   1:  PR[91,1] = PR[90,1] + -40.639;
   1:  PR[91,2] = PR[90,2] + 3.831;
   1:L PR[91] R[100]mm/sec CNT100;
   1:  PR[91,1] = PR[90,1] + -40.703;
   1:  PR[91,2] = PR[90,2] + 3.535;
   1:L PR[91] R[100]mm/sec CNT100;
   1:  PR[91,1] = PR[90,1] + -40.740;
   1:  PR[91,2] = PR[90,2] + 3.017;
   1:L PR[91] R[100]mm/sec CNT100;
   1:  PR[91,1] = PR[90,1] + -41.147;
   1:  PR[91,2] = PR[90,2] + -0.477;
   1:L PR[91] R[100]mm/sec CNT100;
   1:  PR[91,1] = PR[90,1] + -41.119;
   1:  PR[91,2] = PR[90,2] + -0.869;
   1:L PR[91] R[100]mm/sec CNT100;
   1:  PR[91,1] = PR[90,1] + -40.715;
   1:  PR[91,2] = PR[90,2] + -4.331;
   1:L PR[91] R[100]mm/sec CNT100;
   1:  PR[91,1] = PR[90,1] + -40.638;
   1:  PR[91,2] = PR[90,2] + -4.679;
   1:L PR[91] R[100]mm/sec CNT100;
   1:  PR[91,1] = PR[90,1] + -39.266;
   1:  PR[91,2] = PR[90,2] + -8.416;
   1:L PR[91] R[100]mm/sec CNT100;
   1:  PR[91,1] = PR[90,1] + -39.110;
   1:  PR[91,2] = PR[90,2] + -8.700;
   1:L PR[91] R[100]mm/sec CNT100;
   1:  PR[91,1] = PR[90,1] + -37.111;
   1:  PR[91,2] = PR[90,2] + -11.734;
   1:L PR[91] R[100]mm/sec CNT100;
   1:  PR[91,1] = PR[90,1] + -36.935;
   1:  PR[91,2] = PR[90,2] + -11.967;
   1:L PR[91] R[100]mm/sec CNT100;
   1:  PR[91,1] = PR[90,1] + -36.697;
   1:  PR[91,2] = PR[90,2] + -12.203;
   1:L PR[91] R[100]mm/sec CNT100;
   1:  PR[91,1] = PR[90,1] + -33.985;
   1:  PR[91,2] = PR[90,2] + -14.753;
   1:L PR[91] R[100]mm/sec CNT100;
   1:  PR[91,1] = PR[90,1] + -33.873;
   1:  PR[91,2] = PR[90,2] + -14.836;
   1:L PR[91] R[100]mm/sec CNT100;
   1:  PR[91,1] = PR[90,1] + -33.596;
   1:  PR[91,2] = PR[90,2] + -14.985;
   1:L PR[91] R[100]mm/sec CNT100;
   1:  PR[91,1] = PR[90,1] + -30.271;
   1:  PR[91,2] = PR[90,2] + -16.901;
   1:L PR[91] R[100]mm/sec CNT100;
   1:  PR[91,1] = PR[90,1] + -30.216;
   1:  PR[91,2] = PR[90,2] + -16.922;
   1:L PR[91] R[100]mm/sec CNT100;
   1:  PR[91,1] = PR[90,1] + -26.322;
   1:  PR[91,2] = PR[90,2] + -18.082;
   1:L PR[91] R[100]mm/sec CNT100;
   1:  PR[91,1] = PR[90,1] + -22.141;
   1:  PR[91,2] = PR[90,2] + -18.325;
   1:L PR[91] R[100]mm/sec CNT100;
   1:  PR[91,1] = PR[90,1] + -17.967;
   1:  PR[91,2] = PR[90,2] + -17.608;
   1:L PR[91] R[100]mm/sec CNT100;
   1:  PR[91,1] = PR[90,1] + -14.146;
   1:  PR[91,2] = PR[90,2] + -15.991;
   1:L PR[91] R[100]mm/sec CNT100;
   1:  PR[91,1] = PR[90,1] + -13.906;
   1:  PR[91,2] = PR[90,2] + -15.838;
   1:L PR[91] R[100]mm/sec CNT100;
   1:  PR[91,1] = PR[90,1] + -10.813;
   1:  PR[91,2] = PR[90,2] + -13.575;
   1:L PR[91] R[100]mm/sec CNT100;
   1:  PR[91,1] = PR[90,1] + -10.403;
   1:  PR[91,2] = PR[90,2] + -13.158;
   1:L PR[91] R[100]mm/sec CNT100;
   1:  PR[91,1] = PR[90,1] + -8.128;
   1:  PR[91,2] = PR[90,2] + -10.487;
   1:L PR[91] R[100]mm/sec CNT100;
   1:  PR[91,1] = PR[90,1] + -7.743;
   1:  PR[91,2] = PR[90,2] + -9.851;
   1:L PR[91] R[100]mm/sec CNT100;
   1:  PR[91,1] = PR[90,1] + -9.545;
   1:  PR[91,2] = PR[90,2] + -9.686;
   1:L PR[91] R[100]mm/sec CNT100;
   1:  PR[91,1] = PR[90,1] + -5.350;
   1:  PR[91,2] = PR[90,2] + -5.740;
   1:L PR[91] R[100]mm/sec CNT100;
   1:  PR[91,1] = PR[90,1] + -5.315;
   1:  PR[91,2] = PR[90,2] + -5.719;
   1:L PR[91] R[100]mm/sec CNT100;
   1:  PR[91,1] = PR[90,1] + -4.925;
   1:  PR[91,2] = PR[90,2] + -5.085;
   1:L PR[91] R[100]mm/sec CNT100;
   1:  PR[91,1] = PR[90,1] + -2.728;
   1:  PR[91,2] = PR[90,2] + -4.248;
   1:L PR[91] R[100]mm/sec CNT100;
   1:  PR[91,1] = PR[90,1] + 2.325;
   1:L PR[91] R[100]mm/sec CNT100;
   1:  PR[91,1] = PR[90,1] + 3.225;
   1:  PR[91,2] = PR[90,2] + -4.625;
   1:L PR[91] R[100]mm/sec CNT100;
   1:  PR[91,1] = PR[90,1] + 4.250;
   1:  PR[91,2] = PR[90,2] + -5.004;
   1:L PR[91] R[100]mm/sec CNT100;
   1:  PR[91,1] = PR[90,1] + 4.835;
   1:  PR[91,2] = PR[90,2] + -5.693;
   1:L PR[91] R[100]mm/sec CNT100;
   1:  PR[91,1] = PR[90,1] + 4.918;
   1:  PR[91,2] = PR[90,2] + -5.761;
   1:L PR[91] R[100]mm/sec CNT100;
   1:  PR[91,1] = PR[90,1] + 5.507;
   1:  PR[91,2] = PR[90,2] + -6.410;
   1:L PR[91] R[100]mm/sec CNT100;
   1:  PR[91,1] = PR[90,1] + 7.186;
   1:  PR[91,2] = PR[90,2] + -9.719;
   1:L PR[91] R[100]mm/sec CNT100;
   1:  PR[91,1] = PR[90,1] + 7.651;
   1:  PR[91,2] = PR[90,2] + -10.488;
   1:L PR[91] R[100]mm/sec CNT100;
   1:  PR[91,1] = PR[90,1] + 9.927;
   1:  PR[91,2] = PR[90,2] + -13.160;
   1:L PR[91] R[100]mm/sec CNT100;
   1:  PR[91,1] = PR[90,1] + 10.337;
   1:  PR[91,2] = PR[90,2] + -13.578;
   1:L PR[91] R[100]mm/sec CNT100;
   1:  PR[91,1] = PR[90,1] + 13.428;
   1:  PR[91,2] = PR[90,2] + -15.840;
   1:L PR[91] R[100]mm/sec CNT100;
   1:  PR[91,1] = PR[90,1] + 13.668;
   1:  PR[91,2] = PR[90,2] + -15.992;
   1:L PR[91] R[100]mm/sec CNT100;
   1:  PR[91,1] = PR[90,1] + 17.491;
   1:  PR[91,2] = PR[90,2] + -17.609;
   1:L PR[91] R[100]mm/sec CNT100;
   1:  PR[91,1] = PR[90,1] + 21.626;
   1:  PR[91,2] = PR[90,2] + -18.322;
   1:L PR[91] R[100]mm/sec CNT100;
   1:  PR[91,1] = PR[90,1] + 25.845;
   1:  PR[91,2] = PR[90,2] + -18.081;
   1:L PR[91] R[100]mm/sec CNT100;
   1:  PR[91,1] = PR[90,1] + 29.738;
   1:  PR[91,2] = PR[90,2] + -16.921;
   1:L PR[91] R[100]mm/sec CNT100;
   1:  PR[91,1] = PR[90,1] + 29.796;
   1:  PR[91,2] = PR[90,2] + -16.899;
   1:L PR[91] R[100]mm/sec CNT100;
   1:  PR[91,1] = PR[90,1] + 33.369;
   1:  PR[91,2] = PR[90,2] + -14.854;
   1:L PR[91] R[100]mm/sec CNT100;
   1:  PR[91,1] = PR[90,1] + 33.480;
   1:  PR[91,2] = PR[90,2] + -14.772;
   1:L PR[91] R[100]mm/sec CNT100;
   1:  PR[91,1] = PR[90,1] + 33.701;
   1:  PR[91,2] = PR[90,2] + -14.553;
   1:L PR[91] R[100]mm/sec CNT100;
   1:  PR[91,1] = PR[90,1] + 36.475;
   1:  PR[91,2] = PR[90,2] + -11.941;
   1:L PR[91] R[100]mm/sec CNT100;
   1:  PR[91,1] = PR[90,1] + 36.631;
   1:  PR[91,2] = PR[90,2] + -11.732;
   1:L PR[91] R[100]mm/sec CNT100;
   1:  PR[91,1] = PR[90,1] + 38.630;
   1:  PR[91,2] = PR[90,2] + -8.699;
   1:L PR[91] R[100]mm/sec CNT100;
   1:  PR[91,1] = PR[90,1] + 38.791;
   1:  PR[91,2] = PR[90,2] + -8.407;
   1:L PR[91] R[100]mm/sec CNT100;
   1:  PR[91,1] = PR[90,1] + 38.939;
   1:  PR[91,2] = PR[90,2] + -8.013;
   1:L PR[91] R[100]mm/sec CNT100;
   1:  PR[91,1] = PR[90,1] + 40.159;
   1:  PR[91,2] = PR[90,2] + -4.682;
   1:L PR[91] R[100]mm/sec CNT100;
   1:  PR[91,1] = PR[90,1] + 40.223;
   1:  PR[91,2] = PR[90,2] + -4.386;
   1:L PR[91] R[100]mm/sec CNT100;
   1:  PR[91,1] = PR[90,1] + 40.261;
   1:  PR[91,2] = PR[90,2] + -3.867;
   1:L PR[91] R[100]mm/sec CNT100;
   1:  PR[91,1] = PR[90,1] + 40.667;
   1:  PR[91,2] = PR[90,2] + -0.370;
   1:L PR[91] R[100]mm/sec CNT100;
   1:  PR[91,1] = PR[90,1] + 40.639;
   1:  PR[91,2] = PR[90,2] + 0.022;
   1:L PR[91] R[100]mm/sec CNT100;
   1:  PR[91,1] = PR[90,1] + 40.235;
   1:  PR[91,2] = PR[90,2] + 3.486;
   1:L PR[91] R[100]mm/sec CNT100;
   1:  PR[91,1] = PR[90,1] + 40.159;
   1:  PR[91,2] = PR[90,2] + 3.833;
   1:L PR[91] R[100]mm/sec CNT100;
   1:  PR[91,1] = PR[90,1] + 38.787;
   1:  PR[91,2] = PR[90,2] + 7.567;
   1:L PR[91] R[100]mm/sec CNT100;
   1:  PR[91,1] = PR[90,1] + 38.631;
   1:  PR[91,2] = PR[90,2] + 7.852;
   1:L PR[91] R[100]mm/sec CNT100;
   1:  PR[91,1] = PR[90,1] + 36.632;
   1:  PR[91,2] = PR[90,2] + 10.885;
   1:L PR[91] R[100]mm/sec CNT100;
   1:  PR[91,1] = PR[90,1] + 36.456;
   1:  PR[91,2] = PR[90,2] + 11.118;
   1:L PR[91] R[100]mm/sec CNT100;
   1:  PR[91,1] = PR[90,1] + 36.218;
   1:  PR[91,2] = PR[90,2] + 11.354;
   1:L PR[91] R[100]mm/sec CNT100;
   1:  PR[91,1] = PR[90,1] + 33.507;
   1:  PR[91,2] = PR[90,2] + 13.905;
   1:L PR[91] R[100]mm/sec CNT100;
   1:  PR[91,1] = PR[90,1] + 33.394;
   1:  PR[91,2] = PR[90,2] + 13.989;
   1:L PR[91] R[100]mm/sec CNT100;
   1:  PR[91,1] = PR[90,1] + 33.118;
   1:  PR[91,2] = PR[90,2] + 14.138;
   1:L PR[91] R[100]mm/sec CNT100;
   1:  PR[91,1] = PR[90,1] + 29.794;
   1:  PR[91,2] = PR[90,2] + 16.053;
   1:L PR[91] R[100]mm/sec CNT100;
   1:  PR[91,1] = PR[90,1] + 29.738;
   1:  PR[91,2] = PR[90,2] + 16.073;
   1:L PR[91] R[100]mm/sec CNT100;
   1:  PR[91,1] = PR[90,1] + 25.840;
   1:  PR[91,2] = PR[90,2] + 17.235;
   1:L PR[91] R[100]mm/sec CNT100;
   1:  PR[91,1] = PR[90,1] + 21.627;
   1:  PR[91,2] = PR[90,2] + 17.475;
   1:L PR[91] R[100]mm/sec CNT100;
   1:  PR[91,1] = PR[90,1] + 17.492;
   1:  PR[91,2] = PR[90,2] + 16.762;
   1:L PR[91] R[100]mm/sec CNT100;
   1:  PR[91,1] = PR[90,1] + 13.669;
   1:  PR[91,2] = PR[90,2] + 15.146;
   1:L PR[91] R[100]mm/sec CNT100;
   1:  PR[91,1] = PR[90,1] + 13.430;
   1:  PR[91,2] = PR[90,2] + 14.993;
   1:L PR[91] R[100]mm/sec CNT100;
   1:  PR[91,1] = PR[90,1] + 10.338;
   1:  PR[91,2] = PR[90,2] + 12.732;
   1:L PR[91] R[100]mm/sec CNT100;
   1:  PR[91,1] = PR[90,1] + 9.927;
   1:  PR[91,2] = PR[90,2] + 12.314;
   1:L PR[91] R[100]mm/sec CNT100;
   1:  PR[91,1] = PR[90,1] + 7.650;
   1:  PR[91,2] = PR[90,2] + 9.639;
   1:L PR[91] R[100]mm/sec CNT100;
   1:  PR[91,1] = PR[90,1] + 7.199;
   1:  PR[91,2] = PR[90,2] + 8.897;
   1:L PR[91] R[100]mm/sec CNT100;
   1:  PR[91,1] = PR[90,1] + 5.521;
   1:  PR[91,2] = PR[90,2] + 5.588;
   1:L PR[91] R[100]mm/sec CNT100;
   1:  PR[91,1] = PR[90,1] + 4.973;
   1:  PR[91,2] = PR[90,2] + 4.956;
   1:L PR[91] R[100]mm/sec CNT100;
   1:  PR[91,1] = PR[90,1] + 4.835;
   1:  PR[91,2] = PR[90,2] + 4.871;
   1:L PR[91] R[100]mm/sec CNT100;
   1:  PR[91,1] = PR[90,1] + 4.448;
   1:  PR[91,2] = PR[90,2] + 4.242;
   1:L PR[91] R[100]mm/sec CNT100;
   1:  PR[91,1] = PR[90,1] + 2.263;
   1:  PR[91,2] = PR[90,2] + 3.401;
   1:L PR[91] R[100]mm/sec CNT100;
   1:  PR[91] = PR[90];
   1:  PR[91,1] = PR[90,1] + -2.779;
   1:  PR[91,2] = PR[90,2] + 3.945;
   1:  PR[91,3] = PR[90,3] + 11.895;
   1:L PR[91] R[100]mm/sec CNT100;
   1:  PR[91,1] = PR[90,1] + -4.758;
   1:  PR[91,2] = PR[90,2] + 4.725;
   1:L PR[91] R[100]mm/sec CNT100;
   1:  PR[91,1] = PR[90,1] + -5.390;
   1:  PR[91,2] = PR[90,2] + 5.478;
   1:L PR[91] R[100]mm/sec CNT100;
   1:  PR[91,1] = PR[90,1] + -5.443;
   1:  PR[91,2] = PR[90,2] + 5.521;
   1:L PR[91] R[100]mm/sec CNT100;
   1:  PR[91,1] = PR[90,1] + -5.916;
   1:  PR[91,2] = PR[90,2] + 6.032;
   1:L PR[91] R[100]mm/sec CNT100;
   1:  PR[91,1] = PR[90,1] + -6.700;
   1:  PR[91,2] = PR[90,2] + 7.567;
   1:L PR[91] R[100]mm/sec CNT100;
   1:  PR[91,1] = PR[90,1] + -6.925;
   1:  PR[91,2] = PR[90,2] + 8.038;
   1:L PR[91] R[100]mm/sec CNT100;
   1:  PR[91,1] = PR[90,1] + -8.136;
   1:  PR[91,2] = PR[90,2] + 10.031;
   1:L PR[91] R[100]mm/sec CNT100;
   1:  PR[91,1] = PR[90,1] + -9.464;
   1:  PR[91,2] = PR[90,2] + 11.590;
   1:L PR[91] R[100]mm/sec CNT100;
   1:  PR[91,1] = PR[90,1] + -10.869;
   1:  PR[91,2] = PR[90,2] + 13.017;
   1:L PR[91] R[100]mm/sec CNT100;
   1:  PR[91,1] = PR[90,1] + -12.830;
   1:  PR[91,2] = PR[90,2] + 14.451;
   1:L PR[91] R[100]mm/sec CNT100;
   1:  PR[91,1] = PR[90,1] + -14.219;
   1:  PR[91,2] = PR[90,2] + 15.336;
   1:L PR[91] R[100]mm/sec CNT100;
   1:  PR[91,1] = PR[90,1] + -16.835;
   1:  PR[91,2] = PR[90,2] + 16.442;
   1:L PR[91] R[100]mm/sec CNT100;
   1:  PR[91,1] = PR[90,1] + -18.025;
   1:  PR[91,2] = PR[90,2] + 16.868;
   1:L PR[91] R[100]mm/sec CNT100;
   1:  PR[91,1] = PR[90,1] + -21.222;
   1:  PR[91,2] = PR[90,2] + 17.414;
   1:L PR[91] R[100]mm/sec CNT100;
   1:  PR[91,1] = PR[90,1] + -22.100;
   1:  PR[91,2] = PR[90,2] + 17.520;
   1:L PR[91] R[100]mm/sec CNT100;
   1:  PR[91,1] = PR[90,1] + -25.708;
   1:  PR[91,2] = PR[90,2] + 17.300;
   1:L PR[91] R[100]mm/sec CNT100;
   1:  PR[91,1] = PR[90,1] + -26.240;
   1:  PR[91,2] = PR[90,2] + 17.245;
   1:L PR[91] R[100]mm/sec CNT100;
   1:  PR[91,1] = PR[90,1] + -30.007;
   1:  PR[91,2] = PR[90,2] + 16.115;
   1:L PR[91] R[100]mm/sec CNT100;
   1:  PR[91,1] = PR[90,1] + -30.222;
   1:  PR[91,2] = PR[90,2] + 16.042;
   1:L PR[91] R[100]mm/sec CNT100;
   1:  PR[91,1] = PR[90,1] + -33.862;
   1:  PR[91,2] = PR[90,2] + 13.940;
   1:L PR[91] R[100]mm/sec CNT100;
   1:  PR[91,1] = PR[90,1] + -36.897;
   1:  PR[91,2] = PR[90,2] + 11.090;
   1:L PR[91] R[100]mm/sec CNT100;
   1:  PR[91,1] = PR[90,1] + -39.194;
   1:  PR[91,2] = PR[90,2] + 7.604;
   1:L PR[91] R[100]mm/sec CNT100;
   1:  PR[91,1] = PR[90,1] + -40.607;
   1:  PR[91,2] = PR[90,2] + 3.743;
   1:L PR[91] R[100]mm/sec CNT100;
   1:  PR[91,1] = PR[90,1] + -41.096;
   1:  PR[91,2] = PR[90,2] + -0.424;
   1:L PR[91] R[100]mm/sec CNT100;
   1:  PR[91,1] = PR[90,1] + -40.607;
   1:  PR[91,2] = PR[90,2] + -4.590;
   1:L PR[91] R[100]mm/sec CNT100;
   1:  PR[91,1] = PR[90,1] + -39.177;
   1:  PR[91,2] = PR[90,2] + -8.483;
   1:L PR[91] R[100]mm/sec CNT100;
   1:  PR[91,1] = PR[90,1] + -38.095;
   1:  PR[91,2] = PR[90,2] + -10.124;
   1:L PR[91] R[100]mm/sec CNT100;
   1:  PR[91,1] = PR[90,1] + -36.896;
   1:  PR[91,2] = PR[90,2] + -11.938;
   1:L PR[91] R[100]mm/sec CNT100;
   1:  PR[91,1] = PR[90,1] + -33.860;
   1:  PR[91,2] = PR[90,2] + -14.789;
   1:L PR[91] R[100]mm/sec CNT100;
   1:  PR[91,1] = PR[90,1] + -30.220;
   1:  PR[91,2] = PR[90,2] + -16.890;
   1:L PR[91] R[100]mm/sec CNT100;
   1:  PR[91,1] = PR[90,1] + -30.004;
   1:  PR[91,2] = PR[90,2] + -16.963;
   1:L PR[91] R[100]mm/sec CNT100;
   1:  PR[91,1] = PR[90,1] + -26.236;
   1:  PR[91,2] = PR[90,2] + -18.093;
   1:L PR[91] R[100]mm/sec CNT100;
   1:  PR[91,1] = PR[90,1] + -25.705;
   1:  PR[91,2] = PR[90,2] + -18.147;
   1:L PR[91] R[100]mm/sec CNT100;
   1:  PR[91,1] = PR[90,1] + -22.097;
   1:  PR[91,2] = PR[90,2] + -18.367;
   1:L PR[91] R[100]mm/sec CNT100;
   1:  PR[91,1] = PR[90,1] + -21.219;
   1:  PR[91,2] = PR[90,2] + -18.261;
   1:L PR[91] R[100]mm/sec CNT100;
   1:  PR[91,1] = PR[90,1] + -18.021;
   1:  PR[91,2] = PR[90,2] + -17.714;
   1:L PR[91] R[100]mm/sec CNT100;
   1:  PR[91,1] = PR[90,1] + -16.832;
   1:  PR[91,2] = PR[90,2] + -17.288;
   1:L PR[91] R[100]mm/sec CNT100;
   1:  PR[91,1] = PR[90,1] + -14.216;
   1:  PR[91,2] = PR[90,2] + -16.181;
   1:L PR[91] R[100]mm/sec CNT100;
   1:  PR[91,1] = PR[90,1] + -12.827;
   1:  PR[91,2] = PR[90,2] + -15.297;
   1:L PR[91] R[100]mm/sec CNT100;
   1:  PR[91,1] = PR[90,1] + -10.867;
   1:  PR[91,2] = PR[90,2] + -13.862;
   1:L PR[91] R[100]mm/sec CNT100;
   1:  PR[91,1] = PR[90,1] + -9.462;
   1:  PR[91,2] = PR[90,2] + -12.435;
   1:L PR[91] R[100]mm/sec CNT100;
   1:  PR[91,1] = PR[90,1] + -8.135;
   1:  PR[91,2] = PR[90,2] + -10.876;
   1:L PR[91] R[100]mm/sec CNT100;
   1:  PR[91,1] = PR[90,1] + -7.800;
   1:  PR[91,2] = PR[90,2] + -10.324;
   1:L PR[91] R[100]mm/sec CNT100;
   1:  PR[91,1] = PR[90,1] + -8.623;
   1:  PR[91,2] = PR[90,2] + -10.249;
   1:L PR[91] R[100]mm/sec CNT100;
   1:  PR[91,1] = PR[90,1] + -5.554;
   1:  PR[91,2] = PR[90,2] + -6.446;
   1:L PR[91] R[100]mm/sec CNT100;
   1:  PR[91,1] = PR[90,1] + -5.260;
   1:  PR[91,2] = PR[90,2] + -6.169;
   1:L PR[91] R[100]mm/sec CNT100;
   1:  PR[91,1] = PR[90,1] + -4.930;
   1:  PR[91,2] = PR[90,2] + -5.633;
   1:L PR[91] R[100]mm/sec CNT100;
   1:  PR[91,1] = PR[90,1] + -2.745;
   1:  PR[91,2] = PR[90,2] + -4.793;
   1:L PR[91] R[100]mm/sec CNT100;
   1:  PR[91,1] = PR[90,1] + 2.332;
   1:L PR[91] R[100]mm/sec CNT100;
   1:  PR[91,1] = PR[90,1] + 4.277;
   1:  PR[91,2] = PR[90,2] + -5.577;
   1:L PR[91] R[100]mm/sec CNT100;
   1:  PR[91,1] = PR[90,1] + 4.930;
   1:  PR[91,2] = PR[90,2] + -6.345;
   1:L PR[91] R[100]mm/sec CNT100;
   1:  PR[91,1] = PR[90,1] + 5.045;
   1:  PR[91,2] = PR[90,2] + -6.440;
   1:L PR[91] R[100]mm/sec CNT100;
   1:  PR[91,1] = PR[90,1] + 5.451;
   1:  PR[91,2] = PR[90,2] + -6.887;
   1:L PR[91] R[100]mm/sec CNT100;
   1:  PR[91,1] = PR[90,1] + 6.016;
   1:  PR[91,2] = PR[90,2] + -7.992;
   1:L PR[91] R[100]mm/sec CNT100;
   1:  PR[91,1] = PR[90,1] + 6.411;
   1:  PR[91,2] = PR[90,2] + -8.813;
   1:L PR[91] R[100]mm/sec CNT100;
   1:  PR[91,1] = PR[90,1] + 7.657;
   1:  PR[91,2] = PR[90,2] + -10.876;
   1:L PR[91] R[100]mm/sec CNT100;
   1:  PR[91,1] = PR[90,1] + 8.985;
   1:  PR[91,2] = PR[90,2] + -12.435;
   1:L PR[91] R[100]mm/sec CNT100;
   1:  PR[91,1] = PR[90,1] + 10.390;
   1:  PR[91,2] = PR[90,2] + -13.865;
   1:L PR[91] R[100]mm/sec CNT100;
   1:  PR[91,1] = PR[90,1] + 12.349;
   1:  PR[91,2] = PR[90,2] + -15.299;
   1:L PR[91] R[100]mm/sec CNT100;
   1:  PR[91,1] = PR[90,1] + 13.737;
   1:  PR[91,2] = PR[90,2] + -16.182;
   1:L PR[91] R[100]mm/sec CNT100;
   1:  PR[91,1] = PR[90,1] + 16.354;
   1:  PR[91,2] = PR[90,2] + -17.289;
   1:L PR[91] R[100]mm/sec CNT100;
   1:  PR[91,1] = PR[90,1] + 17.544;
   1:  PR[91,2] = PR[90,2] + -17.714;
   1:L PR[91] R[100]mm/sec CNT100;
   1:  PR[91,1] = PR[90,1] + 20.741;
   1:  PR[91,2] = PR[90,2] + -18.261;
   1:L PR[91] R[100]mm/sec CNT100;
   1:  PR[91,1] = PR[90,1] + 21.619;
   1:  PR[91,2] = PR[90,2] + -18.367;
   1:L PR[91] R[100]mm/sec CNT100;
   1:  PR[91,1] = PR[90,1] + 25.227;
   1:  PR[91,2] = PR[90,2] + -18.147;
   1:L PR[91] R[100]mm/sec CNT100;
   1:  PR[91,1] = PR[90,1] + 25.758;
   1:  PR[91,2] = PR[90,2] + -18.092;
   1:L PR[91] R[100]mm/sec CNT100;
   1:  PR[91,1] = PR[90,1] + 29.526;
   1:  PR[91,2] = PR[90,2] + -16.962;
   1:L PR[91] R[100]mm/sec CNT100;
   1:  PR[91,1] = PR[90,1] + 29.742;
   1:  PR[91,2] = PR[90,2] + -16.889;
   1:L PR[91] R[100]mm/sec CNT100;
   1:  PR[91,1] = PR[90,1] + 33.381;
   1:  PR[91,2] = PR[90,2] + -14.789;
   1:L PR[91] R[100]mm/sec CNT100;
   1:  PR[91,1] = PR[90,1] + 36.417;
   1:  PR[91,2] = PR[90,2] + -11.937;
   1:L PR[91] R[100]mm/sec CNT100;
   1:  PR[91,1] = PR[90,1] + 38.698;
   1:  PR[91,2] = PR[90,2] + -8.481;
   1:L PR[91] R[100]mm/sec CNT100;
   1:  PR[91,1] = PR[90,1] + 40.139;
   1:  PR[91,2] = PR[90,2] + -4.562;
   1:L PR[91] R[100]mm/sec CNT100;
   1:  PR[91,1] = PR[90,1] + 40.617;
   1:  PR[91,2] = PR[90,2] + -0.424;
   1:L PR[91] R[100]mm/sec CNT100;
   1:  PR[91,1] = PR[90,1] + 40.138;
   1:  PR[91,2] = PR[90,2] + 3.715;
   1:L PR[91] R[100]mm/sec CNT100;
   1:  PR[91,1] = PR[90,1] + 38.715;
   1:  PR[91,2] = PR[90,2] + 7.603;
   1:L PR[91] R[100]mm/sec CNT100;
   1:  PR[91,1] = PR[90,1] + 36.413;
   1:  PR[91,2] = PR[90,2] + 11.095;
   1:L PR[91] R[100]mm/sec CNT100;
   1:  PR[91,1] = PR[90,1] + 33.361;
   1:  PR[91,2] = PR[90,2] + 13.961;
   1:L PR[91] R[100]mm/sec CNT100;
   1:  PR[91,1] = PR[90,1] + 29.744;
   1:  PR[91,2] = PR[90,2] + 16.041;
   1:L PR[91] R[100]mm/sec CNT100;
   1:  PR[91,1] = PR[90,1] + 29.527;
   1:  PR[91,2] = PR[90,2] + 16.115;
   1:L PR[91] R[100]mm/sec CNT100;
   1:  PR[91,1] = PR[90,1] + 25.759;
   1:  PR[91,2] = PR[90,2] + 17.245;
   1:L PR[91] R[100]mm/sec CNT100;
   1:  PR[91,1] = PR[90,1] + 25.228;
   1:  PR[91,2] = PR[90,2] + 17.300;
   1:L PR[91] R[100]mm/sec CNT100;
   1:  PR[91,1] = PR[90,1] + 21.620;
   1:  PR[91,2] = PR[90,2] + 17.520;
   1:L PR[91] R[100]mm/sec CNT100;
   1:  PR[91,1] = PR[90,1] + 20.742;
   1:  PR[91,2] = PR[90,2] + 17.414;
   1:L PR[91] R[100]mm/sec CNT100;
   1:  PR[91,1] = PR[90,1] + 17.544;
   1:  PR[91,2] = PR[90,2] + 16.867;
   1:L PR[91] R[100]mm/sec CNT100;
   1:  PR[91,1] = PR[90,1] + 16.354;
   1:  PR[91,2] = PR[90,2] + 16.441;
   1:L PR[91] R[100]mm/sec CNT100;
   1:  PR[91,1] = PR[90,1] + 13.738;
   1:  PR[91,2] = PR[90,2] + 15.335;
   1:L PR[91] R[100]mm/sec CNT100;
   1:  PR[91,1] = PR[90,1] + 12.349;
   1:  PR[91,2] = PR[90,2] + 14.451;
   1:L PR[91] R[100]mm/sec CNT100;
   1:  PR[91,1] = PR[90,1] + 10.389;
   1:  PR[91,2] = PR[90,2] + 13.018;
   1:L PR[91] R[100]mm/sec CNT100;
   1:  PR[91,1] = PR[90,1] + 8.984;
   1:  PR[91,2] = PR[90,2] + 11.587;
   1:L PR[91] R[100]mm/sec CNT100;
   1:  PR[91,1] = PR[90,1] + 7.655;
   1:  PR[91,2] = PR[90,2] + 10.026;
   1:L PR[91] R[100]mm/sec CNT100;
   1:  PR[91,1] = PR[90,1] + 7.311;
   1:  PR[91,2] = PR[90,2] + 9.460;
   1:L PR[91] R[100]mm/sec CNT100;
   1:  PR[91,1] = PR[90,1] + 8.315;
   1:  PR[91,2] = PR[90,2] + 9.364;
   1:L PR[91] R[100]mm/sec CNT100;
   1:  PR[91,1] = PR[90,1] + 4.767;
   1:  PR[91,2] = PR[90,2] + 5.276;
   1:L PR[91] R[100]mm/sec CNT100;
   1:  PR[91,1] = PR[90,1] + 4.742;
   1:  PR[91,2] = PR[90,2] + 5.261;
   1:L PR[91] R[100]mm/sec CNT100;
   1:  PR[91,1] = PR[90,1] + 4.453;
   1:  PR[91,2] = PR[90,2] + 4.791;
   1:L PR[91] R[100]mm/sec CNT100;
   1:  PR[91,1] = PR[90,1] + 2.285;
   1:  PR[91,2] = PR[90,2] + 3.945;
   1:L PR[91] R[100]mm/sec CNT100;
   1:  PR[91] = PR[90];
   1:  PR[91,1] = PR[90,1] + -2.791;
   1:  PR[91,2] = PR[90,2] + 4.490;
   1:  PR[91,3] = PR[90,3] + 13.195;
   1:L PR[91] R[100]mm/sec CNT100;
   1:  PR[91,1] = PR[90,1] + -4.763;
   1:  PR[91,2] = PR[90,2] + 5.272;
   1:L PR[91] R[100]mm/sec CNT100;
   1:  PR[91,1] = PR[90,1] + -5.481;
   1:  PR[91,2] = PR[90,2] + 6.129;
   1:L PR[91] R[100]mm/sec CNT100;
   1:  PR[91,1] = PR[90,1] + -5.784;
   1:  PR[91,2] = PR[90,2] + 6.370;
   1:L PR[91] R[100]mm/sec CNT100;
   1:  PR[91,1] = PR[90,1] + -6.154;
   1:  PR[91,2] = PR[90,2] + 7.148;
   1:L PR[91] R[100]mm/sec CNT100;
   1:  PR[91,1] = PR[90,1] + -8.141;
   1:  PR[91,2] = PR[90,2] + 10.419;
   1:L PR[91] R[100]mm/sec CNT100;
   1:  PR[91,1] = PR[90,1] + -8.522;
   1:  PR[91,2] = PR[90,2] + 10.865;
   1:L PR[91] R[100]mm/sec CNT100;
   1:  PR[91,1] = PR[90,1] + -10.921;
   1:  PR[91,2] = PR[90,2] + 13.303;
   1:L PR[91] R[100]mm/sec CNT100;
   1:  PR[91,1] = PR[90,1] + -11.750;
   1:  PR[91,2] = PR[90,2] + 13.909;
   1:L PR[91] R[100]mm/sec CNT100;
   1:  PR[91,1] = PR[90,1] + -14.288;
   1:  PR[91,2] = PR[90,2] + 15.525;
   1:L PR[91] R[100]mm/sec CNT100;
   1:  PR[91,1] = PR[90,1] + -15.674;
   1:  PR[91,2] = PR[90,2] + 16.112;
   1:L PR[91] R[100]mm/sec CNT100;
   1:  PR[91,1] = PR[90,1] + -18.087;
   1:  PR[91,2] = PR[90,2] + 16.975;
   1:L PR[91] R[100]mm/sec CNT100;
   1:  PR[91,1] = PR[90,1] + -20.039;
   1:  PR[91,2] = PR[90,2] + 17.308;
   1:L PR[91] R[100]mm/sec CNT100;
   1:  PR[91,1] = PR[90,1] + -22.139;
   1:  PR[91,2] = PR[90,2] + 17.562;
   1:L PR[91] R[100]mm/sec CNT100;
   1:  PR[91,1] = PR[90,1] + -24.557;
   1:  PR[91,2] = PR[90,2] + 17.414;
   1:L PR[91] R[100]mm/sec CNT100;
   1:  PR[91,1] = PR[90,1] + -26.246;
   1:  PR[91,2] = PR[90,2] + 17.240;
   1:L PR[91] R[100]mm/sec CNT100;
   1:  PR[91,1] = PR[90,1] + -28.936;
   1:  PR[91,2] = PR[90,2] + 16.433;
   1:L PR[91] R[100]mm/sec CNT100;
   1:  PR[91,1] = PR[90,1] + -30.194;
   1:  PR[91,2] = PR[90,2] + 16.007;
   1:L PR[91] R[100]mm/sec CNT100;
   1:  PR[91,1] = PR[90,1] + -32.904;
   1:  PR[91,2] = PR[90,2] + 14.448;
   1:L PR[91] R[100]mm/sec CNT100;
   1:  PR[91,1] = PR[90,1] + -33.774;
   1:  PR[91,2] = PR[90,2] + 13.915;
   1:L PR[91] R[100]mm/sec CNT100;
   1:  PR[91,1] = PR[90,1] + -36.231;
   1:  PR[91,2] = PR[90,2] + 11.608;
   1:L PR[91] R[100]mm/sec CNT100;
   1:  PR[91,1] = PR[90,1] + -36.787;
   1:  PR[91,2] = PR[90,2] + 11.064;
   1:L PR[91] R[100]mm/sec CNT100;
   1:  PR[91,1] = PR[90,1] + -38.742;
   1:  PR[91,2] = PR[90,2] + 8.105;
   1:L PR[91] R[100]mm/sec CNT100;
   1:  PR[91,1] = PR[90,1] + -39.069;
   1:  PR[91,2] = PR[90,2] + 7.592;
   1:L PR[91] R[100]mm/sec CNT100;
   1:  PR[91,1] = PR[90,1] + -40.327;
   1:  PR[91,2] = PR[90,2] + 4.168;
   1:L PR[91] R[100]mm/sec CNT100;
   1:  PR[91,1] = PR[90,1] + -40.493;
   1:  PR[91,2] = PR[90,2] + 3.706;
   1:L PR[91] R[100]mm/sec CNT100;
   1:  PR[91,1] = PR[90,1] + -40.935;
   1:  PR[91,2] = PR[90,2] + -0.042;
   1:L PR[91] R[100]mm/sec CNT100;
   1:  PR[91,1] = PR[90,1] + -40.996;
   1:  PR[91,2] = PR[90,2] + -0.458;
   1:L PR[91] R[100]mm/sec CNT100;
   1:  PR[91,1] = PR[90,1] + -40.695;
   1:  PR[91,2] = PR[90,2] + -3.019;
   1:L PR[91] R[100]mm/sec CNT100;
   1:  PR[91,1] = PR[90,1] + -40.547;
   1:  PR[91,2] = PR[90,2] + -4.065;
   1:L PR[91] R[100]mm/sec CNT100;
   1:  PR[91,1] = PR[90,1] + -40.491;
   1:  PR[91,2] = PR[90,2] + -4.552;
   1:L PR[91] R[100]mm/sec CNT100;
   1:  PR[91,1] = PR[90,1] + -39.068;
   1:  PR[91,2] = PR[90,2] + -8.441;
   1:L PR[91] R[100]mm/sec CNT100;
   1:  PR[91,1] = PR[90,1] + -38.741;
   1:  PR[91,2] = PR[90,2] + -8.954;
   1:L PR[91] R[100]mm/sec CNT100;
   1:  PR[91,1] = PR[90,1] + -36.786;
   1:  PR[91,2] = PR[90,2] + -11.912;
   1:L PR[91] R[100]mm/sec CNT100;
   1:  PR[91,1] = PR[90,1] + -36.230;
   1:  PR[91,2] = PR[90,2] + -12.457;
   1:L PR[91] R[100]mm/sec CNT100;
   1:  PR[91,1] = PR[90,1] + -33.772;
   1:  PR[91,2] = PR[90,2] + -14.763;
   1:L PR[91] R[100]mm/sec CNT100;
   1:  PR[91,1] = PR[90,1] + -32.902;
   1:  PR[91,2] = PR[90,2] + -15.296;
   1:L PR[91] R[100]mm/sec CNT100;
   1:  PR[91,1] = PR[90,1] + -30.192;
   1:  PR[91,2] = PR[90,2] + -16.855;
   1:L PR[91] R[100]mm/sec CNT100;
   1:  PR[91,1] = PR[90,1] + -28.934;
   1:  PR[91,2] = PR[90,2] + -17.281;
   1:L PR[91] R[100]mm/sec CNT100;
   1:  PR[91,1] = PR[90,1] + -26.244;
   1:  PR[91,2] = PR[90,2] + -18.087;
   1:L PR[91] R[100]mm/sec CNT100;
   1:  PR[91,1] = PR[90,1] + -24.555;
   1:  PR[91,2] = PR[90,2] + -18.262;
   1:L PR[91] R[100]mm/sec CNT100;
   1:  PR[91,1] = PR[90,1] + -22.137;
   1:  PR[91,2] = PR[90,2] + -18.409;
   1:L PR[91] R[100]mm/sec CNT100;
   1:  PR[91,1] = PR[90,1] + -20.037;
   1:  PR[91,2] = PR[90,2] + -18.156;
   1:L PR[91] R[100]mm/sec CNT100;
   1:  PR[91,1] = PR[90,1] + -18.085;
   1:  PR[91,2] = PR[90,2] + -17.822;
   1:L PR[91] R[100]mm/sec CNT100;
   1:  PR[91,1] = PR[90,1] + -15.672;
   1:  PR[91,2] = PR[90,2] + -16.958;
   1:L PR[91] R[100]mm/sec CNT100;
   1:  PR[91,1] = PR[90,1] + -14.286;
   1:  PR[91,2] = PR[90,2] + -16.372;
   1:L PR[91] R[100]mm/sec CNT100;
   1:  PR[91,1] = PR[90,1] + -11.748;
   1:  PR[91,2] = PR[90,2] + -14.755;
   1:L PR[91] R[100]mm/sec CNT100;
   1:  PR[91,1] = PR[90,1] + -10.920;
   1:  PR[91,2] = PR[90,2] + -14.149;
   1:L PR[91] R[100]mm/sec CNT100;
   1:  PR[91,1] = PR[90,1] + -8.521;
   1:  PR[91,2] = PR[90,2] + -11.712;
   1:L PR[91] R[100]mm/sec CNT100;
   1:  PR[91,1] = PR[90,1] + -8.141;
   1:  PR[91,2] = PR[90,2] + -11.266;
   1:L PR[91] R[100]mm/sec CNT100;
   1:  PR[91,1] = PR[90,1] + -6.125;
   1:  PR[91,2] = PR[90,2] + -7.938;
   1:L PR[91] R[100]mm/sec CNT100;
   1:  PR[91,1] = PR[90,1] + -5.883;
   1:  PR[91,2] = PR[90,2] + -7.448;
   1:L PR[91] R[100]mm/sec CNT100;
   1:  PR[91,1] = PR[90,1] + -5.190;
   1:  PR[91,2] = PR[90,2] + -6.590;
   1:L PR[91] R[100]mm/sec CNT100;
   1:  PR[91,1] = PR[90,1] + -5.183;
   1:  PR[91,2] = PR[90,2] + -6.584;
   1:L PR[91] R[100]mm/sec CNT100;
   1:  PR[91,1] = PR[90,1] + -4.935;
   1:  PR[91,2] = PR[90,2] + -6.182;
   1:L PR[91] R[100]mm/sec CNT100;
   1:  PR[91,1] = PR[90,1] + -2.762;
   1:  PR[91,2] = PR[90,2] + -5.337;
   1:L PR[91] R[100]mm/sec CNT100;
   1:  PR[91,1] = PR[90,1] + 2.259;
   1:L PR[91] R[100]mm/sec CNT100;
   1:  PR[91,1] = PR[90,1] + 3.046;
   1:  PR[91,2] = PR[90,2] + -5.620;
   1:L PR[91] R[100]mm/sec CNT100;
   1:  PR[91,1] = PR[90,1] + 4.271;
   1:  PR[91,2] = PR[90,2] + -6.121;
   1:L PR[91] R[100]mm/sec CNT100;
   1:  PR[91,1] = PR[90,1] + 5.396;
   1:  PR[91,2] = PR[90,2] + -7.416;
   1:L PR[91] R[100]mm/sec CNT100;
   1:  PR[91,1] = PR[90,1] + 5.622;
   1:  PR[91,2] = PR[90,2] + -7.885;
   1:L PR[91] R[100]mm/sec CNT100;
   1:  PR[91,1] = PR[90,1] + 7.664;
   1:  PR[91,2] = PR[90,2] + -11.264;
   1:L PR[91] R[100]mm/sec CNT100;
   1:  PR[91,1] = PR[90,1] + 8.043;
   1:  PR[91,2] = PR[90,2] + -11.710;
   1:L PR[91] R[100]mm/sec CNT100;
   1:  PR[91,1] = PR[90,1] + 10.442;
   1:  PR[91,2] = PR[90,2] + -14.152;
   1:L PR[91] R[100]mm/sec CNT100;
   1:  PR[91,1] = PR[90,1] + 11.269;
   1:  PR[91,2] = PR[90,2] + -14.757;
   1:L PR[91] R[100]mm/sec CNT100;
   1:  PR[91,1] = PR[90,1] + 13.807;
   1:  PR[91,2] = PR[90,2] + -16.372;
   1:L PR[91] R[100]mm/sec CNT100;
   1:  PR[91,1] = PR[90,1] + 15.193;
   1:  PR[91,2] = PR[90,2] + -16.959;
   1:L PR[91] R[100]mm/sec CNT100;
   1:  PR[91,1] = PR[90,1] + 17.607;
   1:  PR[91,2] = PR[90,2] + -17.821;
   1:L PR[91] R[100]mm/sec CNT100;
   1:  PR[91,1] = PR[90,1] + 19.558;
   1:  PR[91,2] = PR[90,2] + -18.155;
   1:L PR[91] R[100]mm/sec CNT100;
   1:  PR[91,1] = PR[90,1] + 21.659;
   1:  PR[91,2] = PR[90,2] + -18.409;
   1:L PR[91] R[100]mm/sec CNT100;
   1:  PR[91,1] = PR[90,1] + 24.076;
   1:  PR[91,2] = PR[90,2] + -18.262;
   1:L PR[91] R[100]mm/sec CNT100;
   1:  PR[91,1] = PR[90,1] + 25.765;
   1:  PR[91,2] = PR[90,2] + -18.087;
   1:L PR[91] R[100]mm/sec CNT100;
   1:  PR[91,1] = PR[90,1] + 28.455;
   1:  PR[91,2] = PR[90,2] + -17.280;
   1:L PR[91] R[100]mm/sec CNT100;
   1:  PR[91,1] = PR[90,1] + 29.714;
   1:  PR[91,2] = PR[90,2] + -16.855;
   1:L PR[91] R[100]mm/sec CNT100;
   1:  PR[91,1] = PR[90,1] + 32.424;
   1:  PR[91,2] = PR[90,2] + -15.296;
   1:L PR[91] R[100]mm/sec CNT100;
   1:  PR[91,1] = PR[90,1] + 33.293;
   1:  PR[91,2] = PR[90,2] + -14.764;
   1:L PR[91] R[100]mm/sec CNT100;
   1:  PR[91,1] = PR[90,1] + 35.751;
   1:  PR[91,2] = PR[90,2] + -12.456;
   1:L PR[91] R[100]mm/sec CNT100;
   1:  PR[91,1] = PR[90,1] + 36.306;
   1:  PR[91,2] = PR[90,2] + -11.911;
   1:L PR[91] R[100]mm/sec CNT100;
   1:  PR[91,1] = PR[90,1] + 38.262;
   1:  PR[91,2] = PR[90,2] + -8.951;
   1:L PR[91] R[100]mm/sec CNT100;
   1:  PR[91,1] = PR[90,1] + 38.589;
   1:  PR[91,2] = PR[90,2] + -8.439;
   1:L PR[91] R[100]mm/sec CNT100;
   1:  PR[91,1] = PR[90,1] + 40.014;
   1:  PR[91,2] = PR[90,2] + -4.551;
   1:L PR[91] R[100]mm/sec CNT100;
   1:  PR[91,1] = PR[90,1] + 40.455;
   1:  PR[91,2] = PR[90,2] + -0.807;
   1:L PR[91] R[100]mm/sec CNT100;
   1:  PR[91,1] = PR[90,1] + 40.516;
   1:  PR[91,2] = PR[90,2] + -0.389;
   1:L PR[91] R[100]mm/sec CNT100;
   1:  PR[91,1] = PR[90,1] + 40.215;
   1:  PR[91,2] = PR[90,2] + 2.174;
   1:L PR[91] R[100]mm/sec CNT100;
   1:  PR[91,1] = PR[90,1] + 40.067;
   1:  PR[91,2] = PR[90,2] + 3.221;
   1:L PR[91] R[100]mm/sec CNT100;
   1:  PR[91,1] = PR[90,1] + 40.012;
   1:  PR[91,2] = PR[90,2] + 3.709;
   1:L PR[91] R[100]mm/sec CNT100;
   1:  PR[91,1] = PR[90,1] + 38.589;
   1:  PR[91,2] = PR[90,2] + 7.592;
   1:L PR[91] R[100]mm/sec CNT100;
   1:  PR[91,1] = PR[90,1] + 38.262;
   1:  PR[91,2] = PR[90,2] + 8.104;
   1:L PR[91] R[100]mm/sec CNT100;
   1:  PR[91,1] = PR[90,1] + 36.307;
   1:  PR[91,2] = PR[90,2] + 11.063;
   1:L PR[91] R[100]mm/sec CNT100;
   1:  PR[91,1] = PR[90,1] + 35.750;
   1:  PR[91,2] = PR[90,2] + 11.609;
   1:L PR[91] R[100]mm/sec CNT100;
   1:  PR[91,1] = PR[90,1] + 33.294;
   1:  PR[91,2] = PR[90,2] + 13.916;
   1:L PR[91] R[100]mm/sec CNT100;
   1:  PR[91,1] = PR[90,1] + 32.424;
   1:  PR[91,2] = PR[90,2] + 14.448;
   1:L PR[91] R[100]mm/sec CNT100;
   1:  PR[91,1] = PR[90,1] + 29.714;
   1:  PR[91,2] = PR[90,2] + 16.007;
   1:L PR[91] R[100]mm/sec CNT100;
   1:  PR[91,1] = PR[90,1] + 28.455;
   1:  PR[91,2] = PR[90,2] + 16.433;
   1:L PR[91] R[100]mm/sec CNT100;
   1:  PR[91,1] = PR[90,1] + 25.765;
   1:  PR[91,2] = PR[90,2] + 17.240;
   1:L PR[91] R[100]mm/sec CNT100;
   1:  PR[91,1] = PR[90,1] + 24.076;
   1:  PR[91,2] = PR[90,2] + 17.414;
   1:L PR[91] R[100]mm/sec CNT100;
   1:  PR[91,1] = PR[90,1] + 21.659;
   1:  PR[91,2] = PR[90,2] + 17.562;
   1:L PR[91] R[100]mm/sec CNT100;
   1:  PR[91,1] = PR[90,1] + 19.558;
   1:  PR[91,2] = PR[90,2] + 17.308;
   1:L PR[91] R[100]mm/sec CNT100;
   1:  PR[91,1] = PR[90,1] + 17.606;
   1:  PR[91,2] = PR[90,2] + 16.974;
   1:L PR[91] R[100]mm/sec CNT100;
   1:  PR[91,1] = PR[90,1] + 15.192;
   1:  PR[91,2] = PR[90,2] + 16.111;
   1:L PR[91] R[100]mm/sec CNT100;
   1:  PR[91,1] = PR[90,1] + 13.806;
   1:  PR[91,2] = PR[90,2] + 15.525;
   1:L PR[91] R[100]mm/sec CNT100;
   1:  PR[91,1] = PR[90,1] + 11.268;
   1:  PR[91,2] = PR[90,2] + 13.909;
   1:L PR[91] R[100]mm/sec CNT100;
   1:  PR[91,1] = PR[90,1] + 10.441;
   1:  PR[91,2] = PR[90,2] + 13.304;
   1:L PR[91] R[100]mm/sec CNT100;
   1:  PR[91,1] = PR[90,1] + 8.041;
   1:  PR[91,2] = PR[90,2] + 10.860;
   1:L PR[91] R[100]mm/sec CNT100;
   1:  PR[91,1] = PR[90,1] + 7.660;
   1:  PR[91,2] = PR[90,2] + 10.413;
   1:L PR[91] R[100]mm/sec CNT100;
   1:  PR[91,1] = PR[90,1] + 7.366;
   1:  PR[91,2] = PR[90,2] + 9.928;
   1:L PR[91] R[100]mm/sec CNT100;
   1:  PR[91,1] = PR[90,1] + 7.965;
   1:  PR[91,2] = PR[90,2] + 9.871;
   1:L PR[91] R[100]mm/sec CNT100;
   1:  PR[91,1] = PR[90,1] + 5.150;
   1:  PR[91,2] = PR[90,2] + 6.275;
   1:L PR[91] R[100]mm/sec CNT100;
   1:  PR[91,1] = PR[90,1] + 4.750;
   1:  PR[91,2] = PR[90,2] + 5.813;
   1:L PR[91] R[100]mm/sec CNT100;
   1:  PR[91,1] = PR[90,1] + 4.459;
   1:  PR[91,2] = PR[90,2] + 5.341;
   1:L PR[91] R[100]mm/sec CNT100;
   1:  PR[91,1] = PR[90,1] + 2.306;
   1:  PR[91,2] = PR[90,2] + 4.490;
   1:L PR[91] R[100]mm/sec CNT100;
   1:  PR[91] = PR[90];
   1:  PR[91,1] = PR[90,1] + -2.626;
   1:  PR[91,2] = PR[90,2] + 5.034;
   1:  PR[91,3] = PR[90,3] + 14.495;
   1:L PR[91] R[100]mm/sec CNT100;
   1:  PR[91,1] = PR[90,1] + -4.039;
   1:  PR[91,2] = PR[90,2] + 5.545;
   1:L PR[91] R[100]mm/sec CNT100;
   1:  PR[91,1] = PR[90,1] + -4.601;
   1:  PR[91,2] = PR[90,2] + 5.774;
   1:L PR[91] R[100]mm/sec CNT100;
   1:  PR[91,1] = PR[90,1] + -5.122;
   1:  PR[91,2] = PR[90,2] + 6.272;
   1:L PR[91] R[100]mm/sec CNT100;
   1:  PR[91,1] = PR[90,1] + -5.689;
   1:  PR[91,2] = PR[90,2] + 7.040;
   1:L PR[91] R[100]mm/sec CNT100;
   1:  PR[91,1] = PR[90,1] + -7.767;
   1:  PR[91,2] = PR[90,2] + 10.358;
   1:L PR[91] R[100]mm/sec CNT100;
   1:  PR[91,1] = PR[90,1] + -7.979;
   1:  PR[91,2] = PR[90,2] + 10.649;
   1:L PR[91] R[100]mm/sec CNT100;
   1:  PR[91,1] = PR[90,1] + -10.865;
   1:  PR[91,2] = PR[90,2] + 13.504;
   1:L PR[91] R[100]mm/sec CNT100;
   1:  PR[91,1] = PR[90,1] + -14.354;
   1:  PR[91,2] = PR[90,2] + 15.714;
   1:L PR[91] R[100]mm/sec CNT100;
   1:  PR[91,1] = PR[90,1] + -14.513;
   1:  PR[91,2] = PR[90,2] + 15.781;
   1:L PR[91] R[100]mm/sec CNT100;
   1:  PR[91,1] = PR[90,1] + -18.149;
   1:  PR[91,2] = PR[90,2] + 17.082;
   1:L PR[91] R[100]mm/sec CNT100;
   1:  PR[91,1] = PR[90,1] + -18.855;
   1:  PR[91,2] = PR[90,2] + 17.203;
   1:L PR[91] R[100]mm/sec CNT100;
   1:  PR[91,1] = PR[90,1] + -22.179;
   1:  PR[91,2] = PR[90,2] + 17.603;
   1:L PR[91] R[100]mm/sec CNT100;
   1:  PR[91,1] = PR[90,1] + -23.406;
   1:  PR[91,2] = PR[90,2] + 17.528;
   1:L PR[91] R[100]mm/sec CNT100;
   1:  PR[91,1] = PR[90,1] + -26.252;
   1:  PR[91,2] = PR[90,2] + 17.235;
   1:L PR[91] R[100]mm/sec CNT100;
   1:  PR[91,1] = PR[90,1] + -27.864;
   1:  PR[91,2] = PR[90,2] + 16.751;
   1:L PR[91] R[100]mm/sec CNT100;
   1:  PR[91,1] = PR[90,1] + -30.164;
   1:  PR[91,2] = PR[90,2] + 15.973;
   1:L PR[91] R[100]mm/sec CNT100;
   1:  PR[91,1] = PR[90,1] + -31.951;
   1:  PR[91,2] = PR[90,2] + 14.945;
   1:L PR[91] R[100]mm/sec CNT100;
   1:  PR[91,1] = PR[90,1] + -33.708;
   1:  PR[91,2] = PR[90,2] + 13.868;
   1:L PR[91] R[100]mm/sec CNT100;
   1:  PR[91,1] = PR[90,1] + -35.428;
   1:  PR[91,2] = PR[90,2] + 12.254;
   1:L PR[91] R[100]mm/sec CNT100;
   1:  PR[91,1] = PR[90,1] + -36.691;
   1:  PR[91,2] = PR[90,2] + 11.017;
   1:L PR[91] R[100]mm/sec CNT100;
   1:  PR[91,1] = PR[90,1] + -38.110;
   1:  PR[91,2] = PR[90,2] + 8.869;
   1:L PR[91] R[100]mm/sec CNT100;
   1:  PR[91,1] = PR[90,1] + -38.948;
   1:  PR[91,2] = PR[90,2] + 7.556;
   1:L PR[91] R[100]mm/sec CNT100;
   1:  PR[91,1] = PR[90,1] + -40.358;
   1:  PR[91,2] = PR[90,2] + 3.684;
   1:L PR[91] R[100]mm/sec CNT100;
   1:  PR[91,1] = PR[90,1] + -40.692;
   1:  PR[91,2] = PR[90,2] + 0.857;
   1:L PR[91] R[100]mm/sec CNT100;
   1:  PR[91,1] = PR[90,1] + -40.884;
   1:  PR[91,2] = PR[90,2] + -0.458;
   1:L PR[91] R[100]mm/sec CNT100;
   1:  PR[91,1] = PR[90,1] + -40.831;
   1:  PR[91,2] = PR[90,2] + -0.912;
   1:L PR[91] R[100]mm/sec CNT100;
   1:  PR[91,1] = PR[90,1] + -40.510;
   1:  PR[91,2] = PR[90,2] + -3.181;
   1:L PR[91] R[100]mm/sec CNT100;
   1:  PR[91,1] = PR[90,1] + -40.356;
   1:  PR[91,2] = PR[90,2] + -4.537;
   1:L PR[91] R[100]mm/sec CNT100;
   1:  PR[91,1] = PR[90,1] + -38.947;
   1:  PR[91,2] = PR[90,2] + -8.404;
   1:L PR[91] R[100]mm/sec CNT100;
   1:  PR[91,1] = PR[90,1] + -38.110;
   1:  PR[91,2] = PR[90,2] + -9.717;
   1:L PR[91] R[100]mm/sec CNT100;
   1:  PR[91,1] = PR[90,1] + -36.690;
   1:  PR[91,2] = PR[90,2] + -11.865;
   1:L PR[91] R[100]mm/sec CNT100;
   1:  PR[91,1] = PR[90,1] + -35.427;
   1:  PR[91,2] = PR[90,2] + -13.102;
   1:L PR[91] R[100]mm/sec CNT100;
   1:  PR[91,1] = PR[90,1] + -33.707;
   1:  PR[91,2] = PR[90,2] + -14.716;
   1:L PR[91] R[100]mm/sec CNT100;
   1:  PR[91,1] = PR[90,1] + -31.950;
   1:  PR[91,2] = PR[90,2] + -15.793;
   1:L PR[91] R[100]mm/sec CNT100;
   1:  PR[91,1] = PR[90,1] + -30.163;
   1:  PR[91,2] = PR[90,2] + -16.821;
   1:L PR[91] R[100]mm/sec CNT100;
   1:  PR[91,1] = PR[90,1] + -27.863;
   1:  PR[91,2] = PR[90,2] + -17.599;
   1:L PR[91] R[100]mm/sec CNT100;
   1:  PR[91,1] = PR[90,1] + -26.251;
   1:  PR[91,2] = PR[90,2] + -18.082;
   1:L PR[91] R[100]mm/sec CNT100;
   1:  PR[91,1] = PR[90,1] + -23.405;
   1:  PR[91,2] = PR[90,2] + -18.376;
   1:L PR[91] R[100]mm/sec CNT100;
   1:  PR[91,1] = PR[90,1] + -22.177;
   1:  PR[91,2] = PR[90,2] + -18.451;
   1:L PR[91] R[100]mm/sec CNT100;
   1:  PR[91,1] = PR[90,1] + -18.854;
   1:  PR[91,2] = PR[90,2] + -18.050;
   1:L PR[91] R[100]mm/sec CNT100;
   1:  PR[91,1] = PR[90,1] + -18.148;
   1:  PR[91,2] = PR[90,2] + -17.929;
   1:L PR[91] R[100]mm/sec CNT100;
   1:  PR[91,1] = PR[90,1] + -14.512;
   1:  PR[91,2] = PR[90,2] + -16.628;
   1:L PR[91] R[100]mm/sec CNT100;
   1:  PR[91,1] = PR[90,1] + -14.354;
   1:  PR[91,2] = PR[90,2] + -16.561;
   1:L PR[91] R[100]mm/sec CNT100;
   1:  PR[91,1] = PR[90,1] + -10.893;
   1:  PR[91,2] = PR[90,2] + -14.369;
   1:L PR[91] R[100]mm/sec CNT100;
   1:  PR[91,1] = PR[90,1] + -7.976;
   1:  PR[91,2] = PR[90,2] + -11.492;
   1:L PR[91] R[100]mm/sec CNT100;
   1:  PR[91,1] = PR[90,1] + -7.778;
   1:  PR[91,2] = PR[90,2] + -11.222;
   1:L PR[91] R[100]mm/sec CNT100;
   1:  PR[91,1] = PR[90,1] + -8.179;
   1:  PR[91,2] = PR[90,2] + -11.180;
   1:L PR[91] R[100]mm/sec CNT100;
   1:  PR[91,1] = PR[90,1] + -5.183;
   1:  PR[91,2] = PR[90,2] + -7.196;
   1:L PR[91] R[100]mm/sec CNT100;
   1:  PR[91,1] = PR[90,1] + -4.592;
   1:  PR[91,2] = PR[90,2] + -6.594;
   1:L PR[91] R[100]mm/sec CNT100;
   1:  PR[91,1] = PR[90,1] + -2.639;
   1:  PR[91,2] = PR[90,2] + -5.882;
   1:L PR[91] R[100]mm/sec CNT100;
   1:  PR[91,1] = PR[90,1] + 2.143;
   1:L PR[91] R[100]mm/sec CNT100;
   1:  PR[91,1] = PR[90,1] + 3.540;
   1:  PR[91,2] = PR[90,2] + -6.384;
   1:L PR[91] R[100]mm/sec CNT100;
   1:  PR[91,1] = PR[90,1] + 4.126;
   1:  PR[91,2] = PR[90,2] + -6.622;
   1:L PR[91] R[100]mm/sec CNT100;
   1:  PR[91,1] = PR[90,1] + 4.651;
   1:  PR[91,2] = PR[90,2] + -7.129;
   1:L PR[91] R[100]mm/sec CNT100;
   1:  PR[91,1] = PR[90,1] + 5.209;
   1:  PR[91,2] = PR[90,2] + -7.885;
   1:L PR[91] R[100]mm/sec CNT100;
   1:  PR[91,1] = PR[90,1] + 7.263;
   1:  PR[91,2] = PR[90,2] + -11.160;
   1:L PR[91] R[100]mm/sec CNT100;
   1:  PR[91,1] = PR[90,1] + 7.508;
   1:  PR[91,2] = PR[90,2] + -11.500;
   1:L PR[91] R[100]mm/sec CNT100;
   1:  PR[91,1] = PR[90,1] + 10.387;
   1:  PR[91,2] = PR[90,2] + -14.354;
   1:L PR[91] R[100]mm/sec CNT100;
   1:  PR[91,1] = PR[90,1] + 13.874;
   1:  PR[91,2] = PR[90,2] + -16.561;
   1:L PR[91] R[100]mm/sec CNT100;
   1:  PR[91,1] = PR[90,1] + 14.033;
   1:  PR[91,2] = PR[90,2] + -16.628;
   1:L PR[91] R[100]mm/sec CNT100;
   1:  PR[91,1] = PR[90,1] + 17.669;
   1:  PR[91,2] = PR[90,2] + -17.929;
   1:L PR[91] R[100]mm/sec CNT100;
   1:  PR[91,1] = PR[90,1] + 18.376;
   1:  PR[91,2] = PR[90,2] + -18.049;
   1:L PR[91] R[100]mm/sec CNT100;
   1:  PR[91,1] = PR[90,1] + 21.699;
   1:  PR[91,2] = PR[90,2] + -18.451;
   1:L PR[91] R[100]mm/sec CNT100;
   1:  PR[91,1] = PR[90,1] + 22.926;
   1:  PR[91,2] = PR[90,2] + -18.376;
   1:L PR[91] R[100]mm/sec CNT100;
   1:  PR[91,1] = PR[90,1] + 25.772;
   1:  PR[91,2] = PR[90,2] + -18.082;
   1:L PR[91] R[100]mm/sec CNT100;
   1:  PR[91,1] = PR[90,1] + 27.384;
   1:  PR[91,2] = PR[90,2] + -17.598;
   1:L PR[91] R[100]mm/sec CNT100;
   1:  PR[91,1] = PR[90,1] + 29.684;
   1:  PR[91,2] = PR[90,2] + -16.820;
   1:L PR[91] R[100]mm/sec CNT100;
   1:  PR[91,1] = PR[90,1] + 31.472;
   1:  PR[91,2] = PR[90,2] + -15.792;
   1:L PR[91] R[100]mm/sec CNT100;
   1:  PR[91,1] = PR[90,1] + 33.228;
   1:  PR[91,2] = PR[90,2] + -14.717;
   1:L PR[91] R[100]mm/sec CNT100;
   1:  PR[91,1] = PR[90,1] + 34.947;
   1:  PR[91,2] = PR[90,2] + -13.103;
   1:L PR[91] R[100]mm/sec CNT100;
   1:  PR[91,1] = PR[90,1] + 36.210;
   1:  PR[91,2] = PR[90,2] + -11.864;
   1:L PR[91] R[100]mm/sec CNT100;
   1:  PR[91,1] = PR[90,1] + 37.631;
   1:  PR[91,2] = PR[90,2] + -9.714;
   1:L PR[91] R[100]mm/sec CNT100;
   1:  PR[91,1] = PR[90,1] + 38.468;
   1:  PR[91,2] = PR[90,2] + -8.401;
   1:L PR[91] R[100]mm/sec CNT100;
   1:  PR[91,1] = PR[90,1] + 39.878;
   1:  PR[91,2] = PR[90,2] + -4.537;
   1:L PR[91] R[100]mm/sec CNT100;
   1:  PR[91,1] = PR[90,1] + 40.212;
   1:  PR[91,2] = PR[90,2] + -1.708;
   1:L PR[91] R[100]mm/sec CNT100;
   1:  PR[91,1] = PR[90,1] + 40.405;
   1:  PR[91,2] = PR[90,2] + -0.389;
   1:L PR[91] R[100]mm/sec CNT100;
   1:  PR[91,1] = PR[90,1] + 40.351;
   1:  PR[91,2] = PR[90,2] + 0.066;
   1:L PR[91] R[100]mm/sec CNT100;
   1:  PR[91,1] = PR[90,1] + 40.030;
   1:  PR[91,2] = PR[90,2] + 2.336;
   1:L PR[91] R[100]mm/sec CNT100;
   1:  PR[91,1] = PR[90,1] + 39.876;
   1:  PR[91,2] = PR[90,2] + 3.695;
   1:L PR[91] R[100]mm/sec CNT100;
   1:  PR[91,1] = PR[90,1] + 38.468;
   1:  PR[91,2] = PR[90,2] + 7.554;
   1:L PR[91] R[100]mm/sec CNT100;
   1:  PR[91,1] = PR[90,1] + 37.631;
   1:  PR[91,2] = PR[90,2] + 8.866;
   1:L PR[91] R[100]mm/sec CNT100;
   1:  PR[91,1] = PR[90,1] + 36.210;
   1:  PR[91,2] = PR[90,2] + 11.016;
   1:L PR[91] R[100]mm/sec CNT100;
   1:  PR[91,1] = PR[90,1] + 34.947;
   1:  PR[91,2] = PR[90,2] + 12.256;
   1:L PR[91] R[100]mm/sec CNT100;
   1:  PR[91,1] = PR[90,1] + 33.228;
   1:  PR[91,2] = PR[90,2] + 13.870;
   1:L PR[91] R[100]mm/sec CNT100;
   1:  PR[91,1] = PR[90,1] + 31.471;
   1:  PR[91,2] = PR[90,2] + 14.945;
   1:L PR[91] R[100]mm/sec CNT100;
   1:  PR[91,1] = PR[90,1] + 29.684;
   1:  PR[91,2] = PR[90,2] + 15.973;
   1:L PR[91] R[100]mm/sec CNT100;
   1:  PR[91,1] = PR[90,1] + 27.383;
   1:  PR[91,2] = PR[90,2] + 16.751;
   1:L PR[91] R[100]mm/sec CNT100;
   1:  PR[91,1] = PR[90,1] + 25.771;
   1:  PR[91,2] = PR[90,2] + 17.235;
   1:L PR[91] R[100]mm/sec CNT100;
   1:  PR[91,1] = PR[90,1] + 22.925;
   1:  PR[91,2] = PR[90,2] + 17.529;
   1:L PR[91] R[100]mm/sec CNT100;
   1:  PR[91,1] = PR[90,1] + 21.698;
   1:  PR[91,2] = PR[90,2] + 17.604;
   1:L PR[91] R[100]mm/sec CNT100;
   1:  PR[91,1] = PR[90,1] + 18.374;
   1:  PR[91,2] = PR[90,2] + 17.202;
   1:L PR[91] R[100]mm/sec CNT100;
   1:  PR[91,1] = PR[90,1] + 17.668;
   1:  PR[91,2] = PR[90,2] + 17.081;
   1:L PR[91] R[100]mm/sec CNT100;
   1:  PR[91,1] = PR[90,1] + 14.030;
   1:  PR[91,2] = PR[90,2] + 15.780;
   1:L PR[91] R[100]mm/sec CNT100;
   1:  PR[91,1] = PR[90,1] + 13.872;
   1:  PR[91,2] = PR[90,2] + 15.713;
   1:L PR[91] R[100]mm/sec CNT100;
   1:  PR[91,1] = PR[90,1] + 10.413;
   1:  PR[91,2] = PR[90,2] + 13.523;
   1:L PR[91] R[100]mm/sec CNT100;
   1:  PR[91,1] = PR[90,1] + 7.502;
   1:  PR[91,2] = PR[90,2] + 10.646;
   1:L PR[91] R[100]mm/sec CNT100;
   1:  PR[91,1] = PR[90,1] + 7.271;
   1:  PR[91,2] = PR[90,2] + 10.326;
   1:L PR[91] R[100]mm/sec CNT100;
   1:  PR[91,1] = PR[90,1] + 5.200;
   1:  PR[91,2] = PR[90,2] + 7.021;
   1:L PR[91] R[100]mm/sec CNT100;
   1:  PR[91,1] = PR[90,1] + 4.276;
   1:  PR[91,2] = PR[90,2] + 5.812;
   1:L PR[91] R[100]mm/sec CNT100;
   1:  PR[91,1] = PR[90,1] + 2.158;
   1:  PR[91,2] = PR[90,2] + 5.034;
   1:L PR[91] R[100]mm/sec CNT100;
   1:  PR[91] = PR[90];
   1:  PR[91,1] = PR[90,1] + -2.500;
   1:  PR[91,2] = PR[90,2] + 5.579;
   1:  PR[91,3] = PR[90,3] + 15.795;
   1:L PR[91] R[100]mm/sec CNT100;
   1:  PR[91,1] = PR[90,1] + -3.477;
   1:  PR[91,2] = PR[90,2] + 5.932;
   1:L PR[91] R[100]mm/sec CNT100;
   1:  PR[91,1] = PR[90,1] + -4.424;
   1:  PR[91,2] = PR[90,2] + 6.319;
   1:L PR[91] R[100]mm/sec CNT100;
   1:  PR[91,1] = PR[90,1] + -5.116;
   1:  PR[91,2] = PR[90,2] + 6.980;
   1:L PR[91] R[100]mm/sec CNT100;
   1:  PR[91,1] = PR[90,1] + -5.524;
   1:  PR[91,2] = PR[90,2] + 7.532;
   1:L PR[91] R[100]mm/sec CNT100;
   1:  PR[91,1] = PR[90,1] + -6.752;
   1:  PR[91,2] = PR[90,2] + 9.492;
   1:L PR[91] R[100]mm/sec CNT100;
   1:  PR[91,1] = PR[90,1] + -7.887;
   1:  PR[91,2] = PR[90,2] + 11.044;
   1:L PR[91] R[100]mm/sec CNT100;
   1:  PR[91,1] = PR[90,1] + -9.787;
   1:  PR[91,2] = PR[90,2] + 12.924;
   1:L PR[91] R[100]mm/sec CNT100;
   1:  PR[91,1] = PR[90,1] + -10.761;
   1:  PR[91,2] = PR[90,2] + 13.759;
   1:L PR[91] R[100]mm/sec CNT100;
   1:  PR[91,1] = PR[90,1] + -13.602;
   1:  PR[91,2] = PR[90,2] + 15.516;
   1:L PR[91] R[100]mm/sec CNT100;
   1:  PR[91,1] = PR[90,1] + -14.197;
   1:  PR[91,2] = PR[90,2] + 15.835;
   1:L PR[91] R[100]mm/sec CNT100;
   1:  PR[91,1] = PR[90,1] + -18.011;
   1:  PR[91,2] = PR[90,2] + 17.150;
   1:L PR[91] R[100]mm/sec CNT100;
   1:  PR[91,1] = PR[90,1] + -18.047;
   1:  PR[91,2] = PR[90,2] + 17.160;
   1:L PR[91] R[100]mm/sec CNT100;
   1:  PR[91,1] = PR[90,1] + -22.213;
   1:  PR[91,2] = PR[90,2] + 17.645;
   1:L PR[91] R[100]mm/sec CNT100;
   1:  PR[91,1] = PR[90,1] + -22.255;
   1:  PR[91,2] = PR[90,2] + 17.643;
   1:L PR[91] R[100]mm/sec CNT100;
   1:  PR[91,1] = PR[90,1] + -26.259;
   1:  PR[91,2] = PR[90,2] + 17.230;
   1:L PR[91] R[100]mm/sec CNT100;
   1:  PR[91,1] = PR[90,1] + -26.793;
   1:  PR[91,2] = PR[90,2] + 17.069;
   1:L PR[91] R[100]mm/sec CNT100;
   1:  PR[91,1] = PR[90,1] + -30.134;
   1:  PR[91,2] = PR[90,2] + 15.939;
   1:L PR[91] R[100]mm/sec CNT100;
   1:  PR[91,1] = PR[90,1] + -30.998;
   1:  PR[91,2] = PR[90,2] + 15.442;
   1:L PR[91] R[100]mm/sec CNT100;
   1:  PR[91,1] = PR[90,1] + -33.643;
   1:  PR[91,2] = PR[90,2] + 13.821;
   1:L PR[91] R[100]mm/sec CNT100;
   1:  PR[91,1] = PR[90,1] + -34.624;
   1:  PR[91,2] = PR[90,2] + 12.900;
   1:L PR[91] R[100]mm/sec CNT100;
   1:  PR[91,1] = PR[90,1] + -36.594;
   1:  PR[91,2] = PR[90,2] + 10.971;
   1:L PR[91] R[100]mm/sec CNT100;
   1:  PR[91,1] = PR[90,1] + -37.480;
   1:  PR[91,2] = PR[90,2] + 9.631;
   1:L PR[91] R[100]mm/sec CNT100;
   1:  PR[91,1] = PR[90,1] + -38.826;
   1:  PR[91,2] = PR[90,2] + 7.518;
   1:L PR[91] R[100]mm/sec CNT100;
   1:  PR[91,1] = PR[90,1] + -40.223;
   1:  PR[91,2] = PR[90,2] + 3.669;
   1:L PR[91] R[100]mm/sec CNT100;
   1:  PR[91,1] = PR[90,1] + -40.449;
   1:  PR[91,2] = PR[90,2] + 1.756;
   1:L PR[91] R[100]mm/sec CNT100;
   1:  PR[91,1] = PR[90,1] + -40.672;
   1:  PR[91,2] = PR[90,2] + 0.230;
   1:L PR[91] R[100]mm/sec CNT100;
   1:  PR[91,1] = PR[90,1] + -40.743;
   1:  PR[91,2] = PR[90,2] + -0.391;
   1:L PR[91] R[100]mm/sec CNT100;
   1:  PR[91,1] = PR[90,1] + -40.473;
   1:  PR[91,2] = PR[90,2] + -2.296;
   1:L PR[91] R[100]mm/sec CNT100;
   1:  PR[91,1] = PR[90,1] + -40.221;
   1:  PR[91,2] = PR[90,2] + -4.522;
   1:L PR[91] R[100]mm/sec CNT100;
   1:  PR[91,1] = PR[90,1] + -38.826;
   1:  PR[91,2] = PR[90,2] + -8.366;
   1:L PR[91] R[100]mm/sec CNT100;
   1:  PR[91,1] = PR[90,1] + -37.479;
   1:  PR[91,2] = PR[90,2] + -10.479;
   1:L PR[91] R[100]mm/sec CNT100;
   1:  PR[91,1] = PR[90,1] + -36.594;
   1:  PR[91,2] = PR[90,2] + -11.819;
   1:L PR[91] R[100]mm/sec CNT100;
   1:  PR[91,1] = PR[90,1] + -34.624;
   1:  PR[91,2] = PR[90,2] + -13.748;
   1:L PR[91] R[100]mm/sec CNT100;
   1:  PR[91,1] = PR[90,1] + -33.642;
   1:  PR[91,2] = PR[90,2] + -14.669;
   1:L PR[91] R[100]mm/sec CNT100;
   1:  PR[91,1] = PR[90,1] + -30.998;
   1:  PR[91,2] = PR[90,2] + -16.289;
   1:L PR[91] R[100]mm/sec CNT100;
   1:  PR[91,1] = PR[90,1] + -30.133;
   1:  PR[91,2] = PR[90,2] + -16.787;
   1:L PR[91] R[100]mm/sec CNT100;
   1:  PR[91,1] = PR[90,1] + -26.792;
   1:  PR[91,2] = PR[90,2] + -17.917;
   1:L PR[91] R[100]mm/sec CNT100;
   1:  PR[91,1] = PR[90,1] + -26.258;
   1:  PR[91,2] = PR[90,2] + -18.077;
   1:L PR[91] R[100]mm/sec CNT100;
   1:  PR[91,1] = PR[90,1] + -22.255;
   1:  PR[91,2] = PR[90,2] + -18.490;
   1:L PR[91] R[100]mm/sec CNT100;
   1:  PR[91,1] = PR[90,1] + -22.212;
   1:  PR[91,2] = PR[90,2] + -18.493;
   1:L PR[91] R[100]mm/sec CNT100;
   1:  PR[91,1] = PR[90,1] + -18.047;
   1:  PR[91,2] = PR[90,2] + -18.007;
   1:L PR[91] R[100]mm/sec CNT100;
   1:  PR[91,1] = PR[90,1] + -18.010;
   1:  PR[91,2] = PR[90,2] + -17.997;
   1:L PR[91] R[100]mm/sec CNT100;
   1:  PR[91,1] = PR[90,1] + -14.196;
   1:  PR[91,2] = PR[90,2] + -16.682;
   1:L PR[91] R[100]mm/sec CNT100;
   1:  PR[91,1] = PR[90,1] + -13.600;
   1:  PR[91,2] = PR[90,2] + -16.363;
   1:L PR[91] R[100]mm/sec CNT100;
   1:  PR[91,1] = PR[90,1] + -10.759;
   1:  PR[91,2] = PR[90,2] + -14.605;
   1:L PR[91] R[100]mm/sec CNT100;
   1:  PR[91,1] = PR[90,1] + -9.785;
   1:  PR[91,2] = PR[90,2] + -13.769;
   1:L PR[91] R[100]mm/sec CNT100;
   1:  PR[91,1] = PR[90,1] + -7.883;
   1:  PR[91,2] = PR[90,2] + -11.887;
   1:L PR[91] R[100]mm/sec CNT100;
   1:  PR[91,1] = PR[90,1] + -7.744;
   1:  PR[91,2] = PR[90,2] + -11.698;
   1:L PR[91] R[100]mm/sec CNT100;
   1:  PR[91,1] = PR[90,1] + -8.569;
   1:  PR[91,2] = PR[90,2] + -11.610;
   1:L PR[91] R[100]mm/sec CNT100;
   1:  PR[91,1] = PR[90,1] + -4.670;
   1:  PR[91,2] = PR[90,2] + -7.382;
   1:L PR[91] R[100]mm/sec CNT100;
   1:  PR[91,1] = PR[90,1] + -4.016;
   1:  PR[91,2] = PR[90,2] + -6.942;
   1:L PR[91] R[100]mm/sec CNT100;
   1:  PR[91,1] = PR[90,1] + -3.653;
   1:  PR[91,2] = PR[90,2] + -6.854;
   1:L PR[91] R[100]mm/sec CNT100;
   1:  PR[91,1] = PR[90,1] + -3.522;
   1:  PR[91,2] = PR[90,2] + -6.796;
   1:L PR[91] R[100]mm/sec CNT100;
   1:  PR[91,1] = PR[90,1] + -2.508;
   1:  PR[91,2] = PR[90,2] + -6.426;
   1:L PR[91] R[100]mm/sec CNT100;
   1:  PR[91,1] = PR[90,1] + 2.026;
   1:L PR[91] R[100]mm/sec CNT100;
   1:  PR[91,1] = PR[90,1] + 2.911;
   1:  PR[91,2] = PR[90,2] + -6.744;
   1:L PR[91] R[100]mm/sec CNT100;
   1:  PR[91,1] = PR[90,1] + 3.951;
   1:  PR[91,2] = PR[90,2] + -7.167;
   1:L PR[91] R[100]mm/sec CNT100;
   1:  PR[91,1] = PR[90,1] + 4.664;
   1:  PR[91,2] = PR[90,2] + -7.855;
   1:L PR[91] R[100]mm/sec CNT100;
   1:  PR[91,1] = PR[90,1] + 5.048;
   1:  PR[91,2] = PR[90,2] + -8.376;
   1:L PR[91] R[100]mm/sec CNT100;
   1:  PR[91,1] = PR[90,1] + 6.178;
   1:  PR[91,2] = PR[90,2] + -10.177;
   1:L PR[91] R[100]mm/sec CNT100;
   1:  PR[91,1] = PR[90,1] + 7.417;
   1:  PR[91,2] = PR[90,2] + -11.897;
   1:L PR[91] R[100]mm/sec CNT100;
   1:  PR[91,1] = PR[90,1] + 9.311;
   1:  PR[91,2] = PR[90,2] + -13.775;
   1:L PR[91] R[100]mm/sec CNT100;
   1:  PR[91,1] = PR[90,1] + 10.283;
   1:  PR[91,2] = PR[90,2] + -14.610;
   1:L PR[91] R[100]mm/sec CNT100;
   1:  PR[91,1] = PR[90,1] + 13.122;
   1:  PR[91,2] = PR[90,2] + -16.365;
   1:L PR[91] R[100]mm/sec CNT100;
   1:  PR[91,1] = PR[90,1] + 13.717;
   1:  PR[91,2] = PR[90,2] + -16.682;
   1:L PR[91] R[100]mm/sec CNT100;
   1:  PR[91,1] = PR[90,1] + 17.532;
   1:  PR[91,2] = PR[90,2] + -17.997;
   1:L PR[91] R[100]mm/sec CNT100;
   1:  PR[91,1] = PR[90,1] + 17.562;
   1:  PR[91,2] = PR[90,2] + -18.005;
   1:L PR[91] R[100]mm/sec CNT100;
   1:  PR[91,1] = PR[90,1] + 19.499;
   1:  PR[91,2] = PR[90,2] + -18.222;
   1:L PR[91] R[100]mm/sec CNT100;
   1:  PR[91,1] = PR[90,1] + 21.738;
   1:  PR[91,2] = PR[90,2] + -18.493;
   1:L PR[91] R[100]mm/sec CNT100;
   1:  PR[91,1] = PR[90,1] + 21.775;
   1:  PR[91,2] = PR[90,2] + -18.490;
   1:L PR[91] R[100]mm/sec CNT100;
   1:  PR[91,1] = PR[90,1] + 25.779;
   1:  PR[91,2] = PR[90,2] + -18.077;
   1:L PR[91] R[100]mm/sec CNT100;
   1:  PR[91,1] = PR[90,1] + 26.313;
   1:  PR[91,2] = PR[90,2] + -17.916;
   1:L PR[91] R[100]mm/sec CNT100;
   1:  PR[91,1] = PR[90,1] + 29.654;
   1:  PR[91,2] = PR[90,2] + -16.786;
   1:L PR[91] R[100]mm/sec CNT100;
   1:  PR[91,1] = PR[90,1] + 30.519;
   1:  PR[91,2] = PR[90,2] + -16.289;
   1:L PR[91] R[100]mm/sec CNT100;
   1:  PR[91,1] = PR[90,1] + 33.163;
   1:  PR[91,2] = PR[90,2] + -14.670;
   1:L PR[91] R[100]mm/sec CNT100;
   1:  PR[91,1] = PR[90,1] + 34.143;
   1:  PR[91,2] = PR[90,2] + -13.749;
   1:L PR[91] R[100]mm/sec CNT100;
   1:  PR[91,1] = PR[90,1] + 36.114;
   1:  PR[91,2] = PR[90,2] + -11.816;
   1:L PR[91] R[100]mm/sec CNT100;
   1:  PR[91,1] = PR[90,1] + 37.000;
   1:  PR[91,2] = PR[90,2] + -10.476;
   1:L PR[91] R[100]mm/sec CNT100;
   1:  PR[91,1] = PR[90,1] + 38.347;
   1:  PR[91,2] = PR[90,2] + -8.364;
   1:L PR[91] R[100]mm/sec CNT100;
   1:  PR[91,1] = PR[90,1] + 39.743;
   1:  PR[91,2] = PR[90,2] + -4.524;
   1:L PR[91] R[100]mm/sec CNT100;
   1:  PR[91,1] = PR[90,1] + 39.969;
   1:  PR[91,2] = PR[90,2] + -2.610;
   1:L PR[91] R[100]mm/sec CNT100;
   1:  PR[91,1] = PR[90,1] + 40.192;
   1:  PR[91,2] = PR[90,2] + -1.080;
   1:L PR[91] R[100]mm/sec CNT100;
   1:  PR[91,1] = PR[90,1] + 40.263;
   1:  PR[91,2] = PR[90,2] + -0.457;
   1:L PR[91] R[100]mm/sec CNT100;
   1:  PR[91,1] = PR[90,1] + 39.993;
   1:  PR[91,2] = PR[90,2] + 1.451;
   1:L PR[91] R[100]mm/sec CNT100;
   1:  PR[91,1] = PR[90,1] + 39.741;
   1:  PR[91,2] = PR[90,2] + 3.682;
   1:L PR[91] R[100]mm/sec CNT100;
   1:  PR[91,1] = PR[90,1] + 38.347;
   1:  PR[91,2] = PR[90,2] + 7.517;
   1:L PR[91] R[100]mm/sec CNT100;
   1:  PR[91,1] = PR[90,1] + 37.000;
   1:  PR[91,2] = PR[90,2] + 9.629;
   1:L PR[91] R[100]mm/sec CNT100;
   1:  PR[91,1] = PR[90,1] + 36.114;
   1:  PR[91,2] = PR[90,2] + 10.969;
   1:L PR[91] R[100]mm/sec CNT100;
   1:  PR[91,1] = PR[90,1] + 34.143;
   1:  PR[91,2] = PR[90,2] + 12.902;
   1:L PR[91] R[100]mm/sec CNT100;
   1:  PR[91,1] = PR[90,1] + 33.162;
   1:  PR[91,2] = PR[90,2] + 13.823;
   1:L PR[91] R[100]mm/sec CNT100;
   1:  PR[91,1] = PR[90,1] + 30.518;
   1:  PR[91,2] = PR[90,2] + 15.442;
   1:L PR[91] R[100]mm/sec CNT100;
   1:  PR[91,1] = PR[90,1] + 29.653;
   1:  PR[91,2] = PR[90,2] + 15.939;
   1:L PR[91] R[100]mm/sec CNT100;
   1:  PR[91,1] = PR[90,1] + 26.312;
   1:  PR[91,2] = PR[90,2] + 17.069;
   1:L PR[91] R[100]mm/sec CNT100;
   1:  PR[91,1] = PR[90,1] + 25.777;
   1:  PR[91,2] = PR[90,2] + 17.230;
   1:L PR[91] R[100]mm/sec CNT100;
   1:  PR[91,1] = PR[90,1] + 21.773;
   1:  PR[91,2] = PR[90,2] + 17.643;
   1:L PR[91] R[100]mm/sec CNT100;
   1:  PR[91,1] = PR[90,1] + 21.736;
   1:  PR[91,2] = PR[90,2] + 17.645;
   1:L PR[91] R[100]mm/sec CNT100;
   1:  PR[91,1] = PR[90,1] + 19.499;
   1:  PR[91,2] = PR[90,2] + 17.375;
   1:L PR[91] R[100]mm/sec CNT100;
   1:  PR[91,1] = PR[90,1] + 17.560;
   1:  PR[91,2] = PR[90,2] + 17.158;
   1:L PR[91] R[100]mm/sec CNT100;
   1:  PR[91,1] = PR[90,1] + 17.529;
   1:  PR[91,2] = PR[90,2] + 17.149;
   1:L PR[91] R[100]mm/sec CNT100;
   1:  PR[91,1] = PR[90,1] + 13.715;
   1:  PR[91,2] = PR[90,2] + 15.834;
   1:L PR[91] R[100]mm/sec CNT100;
   1:  PR[91,1] = PR[90,1] + 13.120;
   1:  PR[91,2] = PR[90,2] + 15.516;
   1:L PR[91] R[100]mm/sec CNT100;
   1:  PR[91,1] = PR[90,1] + 10.281;
   1:  PR[91,2] = PR[90,2] + 13.761;
   1:L PR[91] R[100]mm/sec CNT100;
   1:  PR[91,1] = PR[90,1] + 9.309;
   1:  PR[91,2] = PR[90,2] + 12.926;
   1:L PR[91] R[100]mm/sec CNT100;
   1:  PR[91,1] = PR[90,1] + 7.413;
   1:  PR[91,2] = PR[90,2] + 11.045;
   1:L PR[91] R[100]mm/sec CNT100;
   1:  PR[91,1] = PR[90,1] + 6.214;
   1:  PR[91,2] = PR[90,2] + 9.390;
   1:L PR[91] R[100]mm/sec CNT100;
   1:  PR[91,1] = PR[90,1] + 5.047;
   1:  PR[91,2] = PR[90,2] + 7.527;
   1:L PR[91] R[100]mm/sec CNT100;
   1:  PR[91,1] = PR[90,1] + 4.652;
   1:  PR[91,2] = PR[90,2] + 6.994;
   1:L PR[91] R[100]mm/sec CNT100;
   1:  PR[91,1] = PR[90,1] + 4.131;
   1:  PR[91,2] = PR[90,2] + 6.494;
   1:L PR[91] R[100]mm/sec CNT100;
   1:  PR[91,1] = PR[90,1] + 3.538;
   1:  PR[91,2] = PR[90,2] + 6.094;
   1:L PR[91] R[100]mm/sec CNT100;
   1:  PR[91,1] = PR[90,1] + 3.172;
   1:  PR[91,2] = PR[90,2] + 6.006;
   1:L PR[91] R[100]mm/sec CNT100;
   1:  PR[91,1] = PR[90,1] + 3.012;
   1:  PR[91,2] = PR[90,2] + 5.936;
   1:L PR[91] R[100]mm/sec CNT100;
   1:  PR[91,1] = PR[90,1] + 2.028;
   1:  PR[91,2] = PR[90,2] + 5.579;
   1:L PR[91] R[100]mm/sec CNT100;
   1:  PR[91] = PR[90];
   1:  PR[91,1] = PR[90,1] + -2.419;
   1:  PR[91,2] = PR[90,2] + 6.124;
   1:  PR[91,3] = PR[90,3] + 17.095;
   1:L PR[91] R[100]mm/sec CNT100;
   1:  PR[91,1] = PR[90,1] + -4.244;
   1:  PR[91,2] = PR[90,2] + 6.860;
   1:L PR[91] R[100]mm/sec CNT100;
   1:  PR[91,1] = PR[90,1] + -5.168;
   1:  PR[91,2] = PR[90,2] + 7.743;
   1:L PR[91] R[100]mm/sec CNT100;
   1:  PR[91,1] = PR[90,1] + -5.729;
   1:  PR[91,2] = PR[90,2] + 8.616;
   1:L PR[91] R[100]mm/sec CNT100;
   1:  PR[91,1] = PR[90,1] + -7.794;
   1:  PR[91,2] = PR[90,2] + 11.439;
   1:L PR[91] R[100]mm/sec CNT100;
   1:  PR[91,1] = PR[90,1] + -8.638;
   1:  PR[91,2] = PR[90,2] + 12.274;
   1:L PR[91] R[100]mm/sec CNT100;
   1:  PR[91,1] = PR[90,1] + -10.708;
   1:  PR[91,2] = PR[90,2] + 14.050;
   1:L PR[91] R[100]mm/sec CNT100;
   1:  PR[91,1] = PR[90,1] + -12.327;
   1:  PR[91,2] = PR[90,2] + 15.051;
   1:L PR[91] R[100]mm/sec CNT100;
   1:  PR[91,1] = PR[90,1] + -14.157;
   1:  PR[91,2] = PR[90,2] + 16.032;
   1:L PR[91] R[100]mm/sec CNT100;
   1:  PR[91,1] = PR[90,1] + -16.668;
   1:  PR[91,2] = PR[90,2] + 16.897;
   1:L PR[91] R[100]mm/sec CNT100;
   1:  PR[91,1] = PR[90,1] + -17.992;
   1:  PR[91,2] = PR[90,2] + 17.275;
   1:L PR[91] R[100]mm/sec CNT100;
   1:  PR[91,1] = PR[90,1] + -21.363;
   1:  PR[91,2] = PR[90,2] + 17.652;
   1:L PR[91] R[100]mm/sec CNT100;
   1:  PR[91,1] = PR[90,1] + -22.049;
   1:  PR[91,2] = PR[90,2] + 17.696;
   1:L PR[91] R[100]mm/sec CNT100;
   1:  PR[91,1] = PR[90,1] + -26.083;
   1:  PR[91,2] = PR[90,2] + 17.259;
   1:L PR[91] R[100]mm/sec CNT100;
   1:  PR[91,1] = PR[90,1] + -26.140;
   1:  PR[91,2] = PR[90,2] + 17.250;
   1:L PR[91] R[100]mm/sec CNT100;
   1:  PR[91,1] = PR[90,1] + -30.073;
   1:  PR[91,2] = PR[90,2] + 15.916;
   1:L PR[91] R[100]mm/sec CNT100;
   1:  PR[91,1] = PR[90,1] + -33.578;
   1:  PR[91,2] = PR[90,2] + 13.773;
   1:L PR[91] R[100]mm/sec CNT100;
   1:  PR[91,1] = PR[90,1] + -33.821;
   1:  PR[91,2] = PR[90,2] + 13.546;
   1:L PR[91] R[100]mm/sec CNT100;
   1:  PR[91,1] = PR[90,1] + -36.498;
   1:  PR[91,2] = PR[90,2] + 10.924;
   1:L PR[91] R[100]mm/sec CNT100;
   1:  PR[91,1] = PR[90,1] + -36.848;
   1:  PR[91,2] = PR[90,2] + 10.394;
   1:L PR[91] R[100]mm/sec CNT100;
   1:  PR[91,1] = PR[90,1] + -38.705;
   1:  PR[91,2] = PR[90,2] + 7.481;
   1:L PR[91] R[100]mm/sec CNT100;
   1:  PR[91,1] = PR[90,1] + -40.088;
   1:  PR[91,2] = PR[90,2] + 3.655;
   1:L PR[91] R[100]mm/sec CNT100;
   1:  PR[91,1] = PR[90,1] + -40.205;
   1:  PR[91,2] = PR[90,2] + 2.656;
   1:L PR[91] R[100]mm/sec CNT100;
   1:  PR[91,1] = PR[90,1] + -40.334;
   1:  PR[91,2] = PR[90,2] + 1.780;
   1:L PR[91] R[100]mm/sec CNT100;
   1:  PR[91,1] = PR[90,1] + -40.581;
   1:  PR[91,2] = PR[90,2] + -0.391;
   1:L PR[91] R[100]mm/sec CNT100;
   1:  PR[91,1] = PR[90,1] + -40.436;
   1:  PR[91,2] = PR[90,2] + -1.412;
   1:L PR[91] R[100]mm/sec CNT100;
   1:  PR[91,1] = PR[90,1] + -40.086;
   1:  PR[91,2] = PR[90,2] + -4.507;
   1:L PR[91] R[100]mm/sec CNT100;
   1:  PR[91,1] = PR[90,1] + -38.705;
   1:  PR[91,2] = PR[90,2] + -8.329;
   1:L PR[91] R[100]mm/sec CNT100;
   1:  PR[91,1] = PR[90,1] + -36.848;
   1:  PR[91,2] = PR[90,2] + -11.241;
   1:L PR[91] R[100]mm/sec CNT100;
   1:  PR[91,1] = PR[90,1] + -36.498;
   1:  PR[91,2] = PR[90,2] + -11.772;
   1:L PR[91] R[100]mm/sec CNT100;
   1:  PR[91,1] = PR[90,1] + -33.820;
   1:  PR[91,2] = PR[90,2] + -14.393;
   1:L PR[91] R[100]mm/sec CNT100;
   1:  PR[91,1] = PR[90,1] + -33.578;
   1:  PR[91,2] = PR[90,2] + -14.621;
   1:L PR[91] R[100]mm/sec CNT100;
   1:  PR[91,1] = PR[90,1] + -30.072;
   1:  PR[91,2] = PR[90,2] + -16.763;
   1:L PR[91] R[100]mm/sec CNT100;
   1:  PR[91,1] = PR[90,1] + -26.140;
   1:  PR[91,2] = PR[90,2] + -18.097;
   1:L PR[91] R[100]mm/sec CNT100;
   1:  PR[91,1] = PR[90,1] + -26.082;
   1:  PR[91,2] = PR[90,2] + -18.106;
   1:L PR[91] R[100]mm/sec CNT100;
   1:  PR[91,1] = PR[90,1] + -22.048;
   1:  PR[91,2] = PR[90,2] + -18.543;
   1:L PR[91] R[100]mm/sec CNT100;
   1:  PR[91,1] = PR[90,1] + -21.361;
   1:  PR[91,2] = PR[90,2] + -18.499;
   1:L PR[91] R[100]mm/sec CNT100;
   1:  PR[91,1] = PR[90,1] + -17.990;
   1:  PR[91,2] = PR[90,2] + -18.122;
   1:L PR[91] R[100]mm/sec CNT100;
   1:  PR[91,1] = PR[90,1] + -16.666;
   1:  PR[91,2] = PR[90,2] + -17.744;
   1:L PR[91] R[100]mm/sec CNT100;
   1:  PR[91,1] = PR[90,1] + -14.154;
   1:  PR[91,2] = PR[90,2] + -16.878;
   1:L PR[91] R[100]mm/sec CNT100;
   1:  PR[91,1] = PR[90,1] + -12.323;
   1:  PR[91,2] = PR[90,2] + -15.895;
   1:L PR[91] R[100]mm/sec CNT100;
   1:  PR[91,1] = PR[90,1] + -10.705;
   1:  PR[91,2] = PR[90,2] + -14.895;
   1:L PR[91] R[100]mm/sec CNT100;
   1:  PR[91,1] = PR[90,1] + -8.634;
   1:  PR[91,2] = PR[90,2] + -13.116;
   1:L PR[91] R[100]mm/sec CNT100;
   1:  PR[91,1] = PR[90,1] + -7.789;
   1:  PR[91,2] = PR[90,2] + -12.281;
   1:L PR[91] R[100]mm/sec CNT100;
   1:  PR[91,1] = PR[90,1] + -7.711;
   1:  PR[91,2] = PR[90,2] + -12.175;
   1:L PR[91] R[100]mm/sec CNT100;
   1:  PR[91,1] = PR[90,1] + -10.464;
   1:  PR[91,2] = PR[90,2] + -11.882;
   1:L PR[91] R[100]mm/sec CNT100;
   1:  PR[91,1] = PR[90,1] + -4.848;
   1:  PR[91,2] = PR[90,2] + -8.309;
   1:L PR[91] R[100]mm/sec CNT100;
   1:  PR[91,1] = PR[90,1] + -4.486;
   1:  PR[91,2] = PR[90,2] + -7.922;
   1:L PR[91] R[100]mm/sec CNT100;
   1:  PR[91,1] = PR[90,1] + -3.788;
   1:  PR[91,2] = PR[90,2] + -7.452;
   1:L PR[91] R[100]mm/sec CNT100;
   1:  PR[91,1] = PR[90,1] + -3.290;
   1:  PR[91,2] = PR[90,2] + -7.331;
   1:L PR[91] R[100]mm/sec CNT100;
   1:  PR[91,1] = PR[90,1] + -2.439;
   1:  PR[91,2] = PR[90,2] + -6.971;
   1:L PR[91] R[100]mm/sec CNT100;
   1:  PR[91,1] = PR[90,1] + 1.949;
   1:L PR[91] R[100]mm/sec CNT100;
   1:  PR[91,1] = PR[90,1] + 3.775;
   1:  PR[91,2] = PR[90,2] + -7.710;
   1:L PR[91] R[100]mm/sec CNT100;
   1:  PR[91,1] = PR[90,1] + 4.734;
   1:  PR[91,2] = PR[90,2] + -8.636;
   1:L PR[91] R[100]mm/sec CNT100;
   1:  PR[91,1] = PR[90,1] + 5.085;
   1:  PR[91,2] = PR[90,2] + -9.183;
   1:L PR[91] R[100]mm/sec CNT100;
   1:  PR[91,1] = PR[90,1] + 7.325;
   1:  PR[91,2] = PR[90,2] + -12.294;
   1:L PR[91] R[100]mm/sec CNT100;
   1:  PR[91,1] = PR[90,1] + 8.163;
   1:  PR[91,2] = PR[90,2] + -13.125;
   1:L PR[91] R[100]mm/sec CNT100;
   1:  PR[91,1] = PR[90,1] + 10.232;
   1:  PR[91,2] = PR[90,2] + -14.902;
   1:L PR[91] R[100]mm/sec CNT100;
   1:  PR[91,1] = PR[90,1] + 11.849;
   1:  PR[91,2] = PR[90,2] + -15.901;
   1:L PR[91] R[100]mm/sec CNT100;
   1:  PR[91,1] = PR[90,1] + 13.678;
   1:  PR[91,2] = PR[90,2] + -16.879;
   1:L PR[91] R[100]mm/sec CNT100;
   1:  PR[91,1] = PR[90,1] + 16.191;
   1:  PR[91,2] = PR[90,2] + -17.745;
   1:L PR[91] R[100]mm/sec CNT100;
   1:  PR[91,1] = PR[90,1] + 17.514;
   1:  PR[91,2] = PR[90,2] + -18.122;
   1:L PR[91] R[100]mm/sec CNT100;
   1:  PR[91,1] = PR[90,1] + 20.884;
   1:  PR[91,2] = PR[90,2] + -18.499;
   1:L PR[91] R[100]mm/sec CNT100;
   1:  PR[91,1] = PR[90,1] + 21.570;
   1:  PR[91,2] = PR[90,2] + -18.543;
   1:L PR[91] R[100]mm/sec CNT100;
   1:  PR[91,1] = PR[90,1] + 25.603;
   1:  PR[91,2] = PR[90,2] + -18.106;
   1:L PR[91] R[100]mm/sec CNT100;
   1:  PR[91,1] = PR[90,1] + 25.660;
   1:  PR[91,2] = PR[90,2] + -18.097;
   1:L PR[91] R[100]mm/sec CNT100;
   1:  PR[91,1] = PR[90,1] + 29.593;
   1:  PR[91,2] = PR[90,2] + -16.763;
   1:L PR[91] R[100]mm/sec CNT100;
   1:  PR[91,1] = PR[90,1] + 33.098;
   1:  PR[91,2] = PR[90,2] + -14.622;
   1:L PR[91] R[100]mm/sec CNT100;
   1:  PR[91,1] = PR[90,1] + 33.340;
   1:  PR[91,2] = PR[90,2] + -14.396;
   1:L PR[91] R[100]mm/sec CNT100;
   1:  PR[91,1] = PR[90,1] + 36.018;
   1:  PR[91,2] = PR[90,2] + -11.769;
   1:L PR[91] R[100]mm/sec CNT100;
   1:  PR[91,1] = PR[90,1] + 36.369;
   1:  PR[91,2] = PR[90,2] + -11.238;
   1:L PR[91] R[100]mm/sec CNT100;
   1:  PR[91,1] = PR[90,1] + 38.226;
   1:  PR[91,2] = PR[90,2] + -8.326;
   1:L PR[91] R[100]mm/sec CNT100;
   1:  PR[91,1] = PR[90,1] + 39.608;
   1:  PR[91,2] = PR[90,2] + -4.510;
   1:L PR[91] R[100]mm/sec CNT100;
   1:  PR[91,1] = PR[90,1] + 39.726;
   1:  PR[91,2] = PR[90,2] + -3.511;
   1:L PR[91] R[100]mm/sec CNT100;
   1:  PR[91,1] = PR[90,1] + 39.854;
   1:  PR[91,2] = PR[90,2] + -2.633;
   1:L PR[91] R[100]mm/sec CNT100;
   1:  PR[91,1] = PR[90,1] + 40.101;
   1:  PR[91,2] = PR[90,2] + -0.457;
   1:L PR[91] R[100]mm/sec CNT100;
   1:  PR[91,1] = PR[90,1] + 39.957;
   1:  PR[91,2] = PR[90,2] + 0.566;
   1:L PR[91] R[100]mm/sec CNT100;
   1:  PR[91,1] = PR[90,1] + 39.606;
   1:  PR[91,2] = PR[90,2] + 3.668;
   1:L PR[91] R[100]mm/sec CNT100;
   1:  PR[91,1] = PR[90,1] + 38.226;
   1:  PR[91,2] = PR[90,2] + 7.479;
   1:L PR[91] R[100]mm/sec CNT100;
   1:  PR[91,1] = PR[90,1] + 36.368;
   1:  PR[91,2] = PR[90,2] + 10.391;
   1:L PR[91] R[100]mm/sec CNT100;
   1:  PR[91,1] = PR[90,1] + 36.017;
   1:  PR[91,2] = PR[90,2] + 10.922;
   1:L PR[91] R[100]mm/sec CNT100;
   1:  PR[91,1] = PR[90,1] + 33.339;
   1:  PR[91,2] = PR[90,2] + 13.549;
   1:L PR[91] R[100]mm/sec CNT100;
   1:  PR[91,1] = PR[90,1] + 33.098;
   1:  PR[91,2] = PR[90,2] + 13.776;
   1:L PR[91] R[100]mm/sec CNT100;
   1:  PR[91,1] = PR[90,1] + 29.592;
   1:  PR[91,2] = PR[90,2] + 15.916;
   1:L PR[91] R[100]mm/sec CNT100;
   1:  PR[91,1] = PR[90,1] + 25.659;
   1:  PR[91,2] = PR[90,2] + 17.250;
   1:L PR[91] R[100]mm/sec CNT100;
   1:  PR[91,1] = PR[90,1] + 25.601;
   1:  PR[91,2] = PR[90,2] + 17.259;
   1:L PR[91] R[100]mm/sec CNT100;
   1:  PR[91,1] = PR[90,1] + 21.568;
   1:  PR[91,2] = PR[90,2] + 17.696;
   1:L PR[91] R[100]mm/sec CNT100;
   1:  PR[91,1] = PR[90,1] + 20.882;
   1:  PR[91,2] = PR[90,2] + 17.652;
   1:L PR[91] R[100]mm/sec CNT100;
   1:  PR[91,1] = PR[90,1] + 17.512;
   1:  PR[91,2] = PR[90,2] + 17.274;
   1:L PR[91] R[100]mm/sec CNT100;
   1:  PR[91,1] = PR[90,1] + 16.189;
   1:  PR[91,2] = PR[90,2] + 16.897;
   1:L PR[91] R[100]mm/sec CNT100;
   1:  PR[91,1] = PR[90,1] + 13.676;
   1:  PR[91,2] = PR[90,2] + 16.031;
   1:L PR[91] R[100]mm/sec CNT100;
   1:  PR[91,1] = PR[90,1] + 11.847;
   1:  PR[91,2] = PR[90,2] + 15.053;
   1:L PR[91] R[100]mm/sec CNT100;
   1:  PR[91,1] = PR[90,1] + 10.231;
   1:  PR[91,2] = PR[90,2] + 14.054;
   1:L PR[91] R[100]mm/sec CNT100;
   1:  PR[91,1] = PR[90,1] + 8.162;
   1:  PR[91,2] = PR[90,2] + 12.276;
   1:L PR[91] R[100]mm/sec CNT100;
   1:  PR[91,1] = PR[90,1] + 7.322;
   1:  PR[91,2] = PR[90,2] + 11.443;
   1:L PR[91] R[100]mm/sec CNT100;
   1:  PR[91,1] = PR[90,1] + 5.149;
   1:  PR[91,2] = PR[90,2] + 8.443;
   1:L PR[91] R[100]mm/sec CNT100;
   1:  PR[91,1] = PR[90,1] + 4.717;
   1:  PR[91,2] = PR[90,2] + 7.769;
   1:L PR[91] R[100]mm/sec CNT100;
   1:  PR[91,1] = PR[90,1] + 3.956;
   1:  PR[91,2] = PR[90,2] + 7.038;
   1:L PR[91] R[100]mm/sec CNT100;
   1:  PR[91,1] = PR[90,1] + 3.312;
   1:  PR[91,2] = PR[90,2] + 6.604;
   1:L PR[91] R[100]mm/sec CNT100;
   1:  PR[91,1] = PR[90,1] + 2.816;
   1:  PR[91,2] = PR[90,2] + 6.484;
   1:L PR[91] R[100]mm/sec CNT100;
   1:  PR[91,1] = PR[90,1] + 1.971;
   1:  PR[91,2] = PR[90,2] + 6.124;
   1:L PR[91] R[100]mm/sec CNT100;
   1:  PR[91] = PR[90];
   1:  PR[91,1] = PR[90,1] + -2.054;
   1:  PR[91,2] = PR[90,2] + 6.668;
   1:  PR[91,3] = PR[90,3] + 18.395;
   1:L PR[91] R[100]mm/sec CNT100;
   1:  PR[91,1] = PR[90,1] + -2.902;
   1:  PR[91,2] = PR[90,2] + 6.873;
   1:L PR[91] R[100]mm/sec CNT100;
   1:  PR[91,1] = PR[90,1] + -3.123;
   1:  PR[91,2] = PR[90,2] + 7.021;
   1:L PR[91] R[100]mm/sec CNT100;
   1:  PR[91,1] = PR[90,1] + -4.145;
   1:  PR[91,2] = PR[90,2] + 7.438;
   1:L PR[91] R[100]mm/sec CNT100;
   1:  PR[91,1] = PR[90,1] + -4.577;
   1:  PR[91,2] = PR[90,2] + 7.907;
   1:L PR[91] R[100]mm/sec CNT100;
   1:  PR[91,1] = PR[90,1] + -4.945;
   1:  PR[91,2] = PR[90,2] + 8.242;
   1:L PR[91] R[100]mm/sec CNT100;
   1:  PR[91,1] = PR[90,1] + -7.624;
   1:  PR[91,2] = PR[90,2] + 11.742;
   1:L PR[91] R[100]mm/sec CNT100;
   1:  PR[91,1] = PR[90,1] + -10.656;
   1:  PR[91,2] = PR[90,2] + 14.340;
   1:L PR[91] R[100]mm/sec CNT100;
   1:  PR[91,1] = PR[90,1] + -11.051;
   1:  PR[91,2] = PR[90,2] + 14.585;
   1:L PR[91] R[100]mm/sec CNT100;
   1:  PR[91,1] = PR[90,1] + -14.117;
   1:  PR[91,2] = PR[90,2] + 16.228;
   1:L PR[91] R[100]mm/sec CNT100;
   1:  PR[91,1] = PR[90,1] + -15.326;
   1:  PR[91,2] = PR[90,2] + 16.645;
   1:L PR[91] R[100]mm/sec CNT100;
   1:  PR[91,1] = PR[90,1] + -17.942;
   1:  PR[91,2] = PR[90,2] + 17.391;
   1:L PR[91] R[100]mm/sec CNT100;
   1:  PR[91,1] = PR[90,1] + -20.012;
   1:  PR[91,2] = PR[90,2] + 17.622;
   1:L PR[91] R[100]mm/sec CNT100;
   1:  PR[91,1] = PR[90,1] + -21.976;
   1:  PR[91,2] = PR[90,2] + 17.749;
   1:L PR[91] R[100]mm/sec CNT100;
   1:  PR[91,1] = PR[90,1] + -24.779;
   1:  PR[91,2] = PR[90,2] + 17.445;
   1:L PR[91] R[100]mm/sec CNT100;
   1:  PR[91,1] = PR[90,1] + -26.033;
   1:  PR[91,2] = PR[90,2] + 17.258;
   1:L PR[91] R[100]mm/sec CNT100;
   1:  PR[91,1] = PR[90,1] + -29.298;
   1:  PR[91,2] = PR[90,2] + 16.148;
   1:L PR[91] R[100]mm/sec CNT100;
   1:  PR[91,1] = PR[90,1] + -29.917;
   1:  PR[91,2] = PR[90,2] + 15.914;
   1:L PR[91] R[100]mm/sec CNT100;
   1:  PR[91,1] = PR[90,1] + -33.288;
   1:  PR[91,2] = PR[90,2] + 13.855;
   1:L PR[91] R[100]mm/sec CNT100;
   1:  PR[91,1] = PR[90,1] + -33.426;
   1:  PR[91,2] = PR[90,2] + 13.766;
   1:L PR[91] R[100]mm/sec CNT100;
   1:  PR[91,1] = PR[90,1] + -36.384;
   1:  PR[91,2] = PR[90,2] + 10.888;
   1:L PR[91] R[100]mm/sec CNT100;
   1:  PR[91,1] = PR[90,1] + -38.585;
   1:  PR[91,2] = PR[90,2] + 7.443;
   1:L PR[91] R[100]mm/sec CNT100;
   1:  PR[91,1] = PR[90,1] + -39.951;
   1:  PR[91,2] = PR[90,2] + 3.642;
   1:L PR[91] R[100]mm/sec CNT100;
   1:  PR[91,1] = PR[90,1] + -40.419;
   1:  PR[91,2] = PR[90,2] + -0.393;
   1:L PR[91] R[100]mm/sec CNT100;
   1:  PR[91,1] = PR[90,1] + -40.400;
   1:  PR[91,2] = PR[90,2] + -0.528;
   1:L PR[91] R[100]mm/sec CNT100;
   1:  PR[91,1] = PR[90,1] + -39.950;
   1:  PR[91,2] = PR[90,2] + -4.493;
   1:L PR[91] R[100]mm/sec CNT100;
   1:  PR[91,1] = PR[90,1] + -38.584;
   1:  PR[91,2] = PR[90,2] + -8.291;
   1:L PR[91] R[100]mm/sec CNT100;
   1:  PR[91,1] = PR[90,1] + -36.836;
   1:  PR[91,2] = PR[90,2] + -11.033;
   1:L PR[91] R[100]mm/sec CNT100;
   1:  PR[91,1] = PR[90,1] + -36.386;
   1:  PR[91,2] = PR[90,2] + -11.733;
   1:L PR[91] R[100]mm/sec CNT100;
   1:  PR[91,1] = PR[90,1] + -33.426;
   1:  PR[91,2] = PR[90,2] + -14.613;
   1:L PR[91] R[100]mm/sec CNT100;
   1:  PR[91,1] = PR[90,1] + -33.288;
   1:  PR[91,2] = PR[90,2] + -14.702;
   1:L PR[91] R[100]mm/sec CNT100;
   1:  PR[91,1] = PR[90,1] + -29.916;
   1:  PR[91,2] = PR[90,2] + -16.761;
   1:L PR[91] R[100]mm/sec CNT100;
   1:  PR[91,1] = PR[90,1] + -29.298;
   1:  PR[91,2] = PR[90,2] + -16.995;
   1:L PR[91] R[100]mm/sec CNT100;
   1:  PR[91,1] = PR[90,1] + -26.032;
   1:  PR[91,2] = PR[90,2] + -18.106;
   1:L PR[91] R[100]mm/sec CNT100;
   1:  PR[91,1] = PR[90,1] + -24.776;
   1:  PR[91,2] = PR[90,2] + -18.293;
   1:L PR[91] R[100]mm/sec CNT100;
   1:  PR[91,1] = PR[90,1] + -21.973;
   1:  PR[91,2] = PR[90,2] + -18.596;
   1:L PR[91] R[100]mm/sec CNT100;
   1:  PR[91,1] = PR[90,1] + -20.008;
   1:  PR[91,2] = PR[90,2] + -18.469;
   1:L PR[91] R[100]mm/sec CNT100;
   1:  PR[91,1] = PR[90,1] + -17.939;
   1:  PR[91,2] = PR[90,2] + -18.238;
   1:L PR[91] R[100]mm/sec CNT100;
   1:  PR[91,1] = PR[90,1] + -15.321;
   1:  PR[91,2] = PR[90,2] + -17.490;
   1:L PR[91] R[100]mm/sec CNT100;
   1:  PR[91,1] = PR[90,1] + -14.112;
   1:  PR[91,2] = PR[90,2] + -17.074;
   1:L PR[91] R[100]mm/sec CNT100;
   1:  PR[91,1] = PR[90,1] + -11.045;
   1:  PR[91,2] = PR[90,2] + -15.428;
   1:L PR[91] R[100]mm/sec CNT100;
   1:  PR[91,1] = PR[90,1] + -10.650;
   1:  PR[91,2] = PR[90,2] + -15.184;
   1:L PR[91] R[100]mm/sec CNT100;
   1:  PR[91,1] = PR[90,1] + -7.619;
   1:  PR[91,2] = PR[90,2] + -12.584;
   1:L PR[91] R[100]mm/sec CNT100;
   1:  PR[91,1] = PR[90,1] + -5.011;
   1:  PR[91,2] = PR[90,2] + -9.174;
   1:L PR[91] R[100]mm/sec CNT100;
   1:  PR[91,1] = PR[90,1] + -4.685;
   1:  PR[91,2] = PR[90,2] + -8.819;
   1:L PR[91] R[100]mm/sec CNT100;
   1:  PR[91,1] = PR[90,1] + -4.572;
   1:  PR[91,2] = PR[90,2] + -8.748;
   1:L PR[91] R[100]mm/sec CNT100;
   1:  PR[91,1] = PR[90,1] + -4.310;
   1:  PR[91,2] = PR[90,2] + -8.467;
   1:L PR[91] R[100]mm/sec CNT100;
   1:  PR[91,1] = PR[90,1] + -3.560;
   1:  PR[91,2] = PR[90,2] + -7.962;
   1:L PR[91] R[100]mm/sec CNT100;
   1:  PR[91,1] = PR[90,1] + -2.957;
   1:  PR[91,2] = PR[90,2] + -7.815;
   1:L PR[91] R[100]mm/sec CNT100;
   1:  PR[91,1] = PR[90,1] + -2.274;
   1:  PR[91,2] = PR[90,2] + -7.515;
   1:L PR[91] R[100]mm/sec CNT100;
   1:  PR[91,1] = PR[90,1] + 1.569;
   1:L PR[91] R[100]mm/sec CNT100;
   1:  PR[91,1] = PR[90,1] + 2.469;
   1:  PR[91,2] = PR[90,2] + -7.732;
   1:L PR[91] R[100]mm/sec CNT100;
   1:  PR[91,1] = PR[90,1] + 2.711;
   1:  PR[91,2] = PR[90,2] + -7.895;
   1:L PR[91] R[100]mm/sec CNT100;
   1:  PR[91,1] = PR[90,1] + 3.668;
   1:  PR[91,2] = PR[90,2] + -8.283;
   1:L PR[91] R[100]mm/sec CNT100;
   1:  PR[91,1] = PR[90,1] + 4.109;
   1:  PR[91,2] = PR[90,2] + -8.761;
   1:L PR[91] R[100]mm/sec CNT100;
   1:  PR[91,1] = PR[90,1] + 4.469;
   1:  PR[91,2] = PR[90,2] + -9.096;
   1:L PR[91] R[100]mm/sec CNT100;
   1:  PR[91,1] = PR[90,1] + 7.149;
   1:  PR[91,2] = PR[90,2] + -12.592;
   1:L PR[91] R[100]mm/sec CNT100;
   1:  PR[91,1] = PR[90,1] + 10.181;
   1:  PR[91,2] = PR[90,2] + -15.194;
   1:L PR[91] R[100]mm/sec CNT100;
   1:  PR[91,1] = PR[90,1] + 10.575;
   1:  PR[91,2] = PR[90,2] + -15.438;
   1:L PR[91] R[100]mm/sec CNT100;
   1:  PR[91,1] = PR[90,1] + 13.639;
   1:  PR[91,2] = PR[90,2] + -17.076;
   1:L PR[91] R[100]mm/sec CNT100;
   1:  PR[91,1] = PR[90,1] + 14.850;
   1:  PR[91,2] = PR[90,2] + -17.493;
   1:L PR[91] R[100]mm/sec CNT100;
   1:  PR[91,1] = PR[90,1] + 17.466;
   1:  PR[91,2] = PR[90,2] + -18.238;
   1:L PR[91] R[100]mm/sec CNT100;
   1:  PR[91,1] = PR[90,1] + 19.535;
   1:  PR[91,2] = PR[90,2] + -18.470;
   1:L PR[91] R[100]mm/sec CNT100;
   1:  PR[91,1] = PR[90,1] + 21.497;
   1:  PR[91,2] = PR[90,2] + -18.596;
   1:L PR[91] R[100]mm/sec CNT100;
   1:  PR[91,1] = PR[90,1] + 24.300;
   1:  PR[91,2] = PR[90,2] + -18.292;
   1:L PR[91] R[100]mm/sec CNT100;
   1:  PR[91,1] = PR[90,1] + 25.554;
   1:  PR[91,2] = PR[90,2] + -18.105;
   1:L PR[91] R[100]mm/sec CNT100;
   1:  PR[91,1] = PR[90,1] + 28.820;
   1:  PR[91,2] = PR[90,2] + -16.994;
   1:L PR[91] R[100]mm/sec CNT100;
   1:  PR[91,1] = PR[90,1] + 29.438;
   1:  PR[91,2] = PR[90,2] + -16.760;
   1:L PR[91] R[100]mm/sec CNT100;
   1:  PR[91,1] = PR[90,1] + 32.810;
   1:  PR[91,2] = PR[90,2] + -14.704;
   1:L PR[91] R[100]mm/sec CNT100;
   1:  PR[91,1] = PR[90,1] + 32.946;
   1:  PR[91,2] = PR[90,2] + -14.615;
   1:L PR[91] R[100]mm/sec CNT100;
   1:  PR[91,1] = PR[90,1] + 35.904;
   1:  PR[91,2] = PR[90,2] + -11.732;
   1:L PR[91] R[100]mm/sec CNT100;
   1:  PR[91,1] = PR[90,1] + 38.106;
   1:  PR[91,2] = PR[90,2] + -8.288;
   1:L PR[91] R[100]mm/sec CNT100;
   1:  PR[91,1] = PR[90,1] + 39.477;
   1:  PR[91,2] = PR[90,2] + -4.483;
   1:L PR[91] R[100]mm/sec CNT100;
   1:  PR[91,1] = PR[90,1] + 39.513;
   1:  PR[91,2] = PR[90,2] + -4.206;
   1:L PR[91] R[100]mm/sec CNT100;
   1:  PR[91,1] = PR[90,1] + 39.939;
   1:  PR[91,2] = PR[90,2] + -0.457;
   1:L PR[91] R[100]mm/sec CNT100;
   1:  PR[91,1] = PR[90,1] + 39.920;
   1:  PR[91,2] = PR[90,2] + -0.319;
   1:L PR[91] R[100]mm/sec CNT100;
   1:  PR[91,1] = PR[90,1] + 39.471;
   1:  PR[91,2] = PR[90,2] + 3.655;
   1:L PR[91] R[100]mm/sec CNT100;
   1:  PR[91,1] = PR[90,1] + 38.105;
   1:  PR[91,2] = PR[90,2] + 7.442;
   1:L PR[91] R[100]mm/sec CNT100;
   1:  PR[91,1] = PR[90,1] + 36.357;
   1:  PR[91,2] = PR[90,2] + 10.182;
   1:L PR[91] R[100]mm/sec CNT100;
   1:  PR[91,1] = PR[90,1] + 35.903;
   1:  PR[91,2] = PR[90,2] + 10.888;
   1:L PR[91] R[100]mm/sec CNT100;
   1:  PR[91,1] = PR[90,1] + 32.945;
   1:  PR[91,2] = PR[90,2] + 13.769;
   1:L PR[91] R[100]mm/sec CNT100;
   1:  PR[91,1] = PR[90,1] + 32.809;
   1:  PR[91,2] = PR[90,2] + 13.857;
   1:L PR[91] R[100]mm/sec CNT100;
   1:  PR[91,1] = PR[90,1] + 29.437;
   1:  PR[91,2] = PR[90,2] + 15.914;
   1:L PR[91] R[100]mm/sec CNT100;
   1:  PR[91,1] = PR[90,1] + 28.819;
   1:  PR[91,2] = PR[90,2] + 16.148;
   1:L PR[91] R[100]mm/sec CNT100;
   1:  PR[91,1] = PR[90,1] + 25.552;
   1:  PR[91,2] = PR[90,2] + 17.258;
   1:L PR[91] R[100]mm/sec CNT100;
   1:  PR[91,1] = PR[90,1] + 24.298;
   1:  PR[91,2] = PR[90,2] + 17.445;
   1:L PR[91] R[100]mm/sec CNT100;
   1:  PR[91,1] = PR[90,1] + 21.496;
   1:  PR[91,2] = PR[90,2] + 17.749;
   1:L PR[91] R[100]mm/sec CNT100;
   1:  PR[91,1] = PR[90,1] + 19.533;
   1:  PR[91,2] = PR[90,2] + 17.623;
   1:L PR[91] R[100]mm/sec CNT100;
   1:  PR[91,1] = PR[90,1] + 17.464;
   1:  PR[91,2] = PR[90,2] + 17.391;
   1:L PR[91] R[100]mm/sec CNT100;
   1:  PR[91,1] = PR[90,1] + 14.848;
   1:  PR[91,2] = PR[90,2] + 16.645;
   1:L PR[91] R[100]mm/sec CNT100;
   1:  PR[91,1] = PR[90,1] + 13.638;
   1:  PR[91,2] = PR[90,2] + 16.228;
   1:L PR[91] R[100]mm/sec CNT100;
   1:  PR[91,1] = PR[90,1] + 10.574;
   1:  PR[91,2] = PR[90,2] + 14.590;
   1:L PR[91] R[100]mm/sec CNT100;
   1:  PR[91,1] = PR[90,1] + 10.180;
   1:  PR[91,2] = PR[90,2] + 14.346;
   1:L PR[91] R[100]mm/sec CNT100;
   1:  PR[91,1] = PR[90,1] + 7.148;
   1:  PR[91,2] = PR[90,2] + 11.743;
   1:L PR[91] R[100]mm/sec CNT100;
   1:  PR[91,1] = PR[90,1] + 4.489;
   1:  PR[91,2] = PR[90,2] + 8.272;
   1:L PR[91] R[100]mm/sec CNT100;
   1:  PR[91,1] = PR[90,1] + 3.789;
   1:  PR[91,2] = PR[90,2] + 7.588;
   1:L PR[91] R[100]mm/sec CNT100;
   1:  PR[91,1] = PR[90,1] + 3.085;
   1:  PR[91,2] = PR[90,2] + 7.114;
   1:L PR[91] R[100]mm/sec CNT100;
   1:  PR[91,1] = PR[90,1] + 2.478;
   1:  PR[91,2] = PR[90,2] + 6.967;
   1:L PR[91] R[100]mm/sec CNT100;
   1:  PR[91,1] = PR[90,1] + 1.792;
   1:  PR[91,2] = PR[90,2] + 6.668;
   1:L PR[91] R[100]mm/sec CNT100;
   1:  PR[91] = PR[90];
   1:  PR[91,1] = PR[90,1] + -1.852;
   1:  PR[91,2] = PR[90,2] + 7.213;
   1:  PR[91,3] = PR[90,3] + 19.695;
   1:L PR[91] R[100]mm/sec CNT100;
   1:  PR[91,1] = PR[90,1] + -2.900;
   1:  PR[91,2] = PR[90,2] + 7.466;
   1:L PR[91] R[100]mm/sec CNT100;
   1:  PR[91,1] = PR[90,1] + -3.209;
   1:  PR[91,2] = PR[90,2] + 7.672;
   1:L PR[91] R[100]mm/sec CNT100;
   1:  PR[91,1] = PR[90,1] + -3.968;
   1:  PR[91,2] = PR[90,2] + 7.982;
   1:L PR[91] R[100]mm/sec CNT100;
   1:  PR[91,1] = PR[90,1] + -4.444;
   1:  PR[91,2] = PR[90,2] + 8.498;
   1:L PR[91] R[100]mm/sec CNT100;
   1:  PR[91,1] = PR[90,1] + -4.711;
   1:  PR[91,2] = PR[90,2] + 8.741;
   1:L PR[91] R[100]mm/sec CNT100;
   1:  PR[91,1] = PR[90,1] + -6.550;
   1:  PR[91,2] = PR[90,2] + 11.145;
   1:L PR[91] R[100]mm/sec CNT100;
   1:  PR[91,1] = PR[90,1] + -7.071;
   1:  PR[91,2] = PR[90,2] + 11.771;
   1:L PR[91] R[100]mm/sec CNT100;
   1:  PR[91,1] = PR[90,1] + -9.859;
   1:  PR[91,2] = PR[90,2] + 14.094;
   1:L PR[91] R[100]mm/sec CNT100;
   1:  PR[91,1] = PR[90,1] + -10.216;
   1:  PR[91,2] = PR[90,2] + 14.409;
   1:L PR[91] R[100]mm/sec CNT100;
   1:  PR[91,1] = PR[90,1] + -10.350;
   1:  PR[91,2] = PR[90,2] + 14.499;
   1:L PR[91] R[100]mm/sec CNT100;
   1:  PR[91,1] = PR[90,1] + -13.487;
   1:  PR[91,2] = PR[90,2] + 16.109;
   1:L PR[91] R[100]mm/sec CNT100;
   1:  PR[91,1] = PR[90,1] + -14.021;
   1:  PR[91,2] = PR[90,2] + 16.395;
   1:L PR[91] R[100]mm/sec CNT100;
   1:  PR[91,1] = PR[90,1] + -17.895;
   1:  PR[91,2] = PR[90,2] + 17.508;
   1:L PR[91] R[100]mm/sec CNT100;
   1:  PR[91,1] = PR[90,1] + -18.661;
   1:  PR[91,2] = PR[90,2] + 17.593;
   1:L PR[91] R[100]mm/sec CNT100;
   1:  PR[91,1] = PR[90,1] + -21.902;
   1:  PR[91,2] = PR[90,2] + 17.802;
   1:L PR[91] R[100]mm/sec CNT100;
   1:  PR[91,1] = PR[90,1] + -23.474;
   1:  PR[91,2] = PR[90,2] + 17.632;
   1:L PR[91] R[100]mm/sec CNT100;
   1:  PR[91,1] = PR[90,1] + -25.927;
   1:  PR[91,2] = PR[90,2] + 17.266;
   1:L PR[91] R[100]mm/sec CNT100;
   1:  PR[91,1] = PR[90,1] + -28.088;
   1:  PR[91,2] = PR[90,2] + 16.531;
   1:L PR[91] R[100]mm/sec CNT100;
   1:  PR[91,1] = PR[90,1] + -29.775;
   1:  PR[91,2] = PR[90,2] + 15.893;
   1:L PR[91] R[100]mm/sec CNT100;
   1:  PR[91,1] = PR[90,1] + -32.210;
   1:  PR[91,2] = PR[90,2] + 14.406;
   1:L PR[91] R[100]mm/sec CNT100;
   1:  PR[91,1] = PR[90,1] + -33.250;
   1:  PR[91,2] = PR[90,2] + 13.731;
   1:L PR[91] R[100]mm/sec CNT100;
   1:  PR[91,1] = PR[90,1] + -35.601;
   1:  PR[91,2] = PR[90,2] + 11.445;
   1:L PR[91] R[100]mm/sec CNT100;
   1:  PR[91,1] = PR[90,1] + -36.166;
   1:  PR[91,2] = PR[90,2] + 10.870;
   1:L PR[91] R[100]mm/sec CNT100;
   1:  PR[91,1] = PR[90,1] + -38.103;
   1:  PR[91,2] = PR[90,2] + 7.858;
   1:L PR[91] R[100]mm/sec CNT100;
   1:  PR[91,1] = PR[90,1] + -38.373;
   1:  PR[91,2] = PR[90,2] + 7.424;
   1:L PR[91] R[100]mm/sec CNT100;
   1:  PR[91,1] = PR[90,1] + -39.748;
   1:  PR[91,2] = PR[90,2] + 3.625;
   1:L PR[91] R[100]mm/sec CNT100;
   1:  PR[91,1] = PR[90,1] + -40.221;
   1:  PR[91,2] = PR[90,2] + -0.424;
   1:L PR[91] R[100]mm/sec CNT100;
   1:  PR[91,1] = PR[90,1] + -39.747;
   1:  PR[91,2] = PR[90,2] + -4.480;
   1:L PR[91] R[100]mm/sec CNT100;
   1:  PR[91,1] = PR[90,1] + -39.644;
   1:  PR[91,2] = PR[90,2] + -4.771;
   1:L PR[91] R[100]mm/sec CNT100;
   1:  PR[91,1] = PR[90,1] + -38.373;
   1:  PR[91,2] = PR[90,2] + -8.270;
   1:L PR[91] R[100]mm/sec CNT100;
   1:  PR[91,1] = PR[90,1] + -38.104;
   1:  PR[91,2] = PR[90,2] + -8.705;
   1:L PR[91] R[100]mm/sec CNT100;
   1:  PR[91,1] = PR[90,1] + -36.166;
   1:  PR[91,2] = PR[90,2] + -11.718;
   1:L PR[91] R[100]mm/sec CNT100;
   1:  PR[91,1] = PR[90,1] + -35.601;
   1:  PR[91,2] = PR[90,2] + -12.292;
   1:L PR[91] R[100]mm/sec CNT100;
   1:  PR[91,1] = PR[90,1] + -33.250;
   1:  PR[91,2] = PR[90,2] + -14.579;
   1:L PR[91] R[100]mm/sec CNT100;
   1:  PR[91,1] = PR[90,1] + -32.208;
   1:  PR[91,2] = PR[90,2] + -15.254;
   1:L PR[91] R[100]mm/sec CNT100;
   1:  PR[91,1] = PR[90,1] + -29.773;
   1:  PR[91,2] = PR[90,2] + -16.741;
   1:L PR[91] R[100]mm/sec CNT100;
   1:  PR[91,1] = PR[90,1] + -28.086;
   1:  PR[91,2] = PR[90,2] + -17.379;
   1:L PR[91] R[100]mm/sec CNT100;
   1:  PR[91,1] = PR[90,1] + -25.925;
   1:  PR[91,2] = PR[90,2] + -18.114;
   1:L PR[91] R[100]mm/sec CNT100;
   1:  PR[91,1] = PR[90,1] + -23.471;
   1:  PR[91,2] = PR[90,2] + -18.479;
   1:L PR[91] R[100]mm/sec CNT100;
   1:  PR[91,1] = PR[90,1] + -21.898;
   1:  PR[91,2] = PR[90,2] + -18.650;
   1:L PR[91] R[100]mm/sec CNT100;
   1:  PR[91,1] = PR[90,1] + -18.655;
   1:  PR[91,2] = PR[90,2] + -18.439;
   1:L PR[91] R[100]mm/sec CNT100;
   1:  PR[91,1] = PR[90,1] + -17.890;
   1:  PR[91,2] = PR[90,2] + -18.354;
   1:L PR[91] R[100]mm/sec CNT100;
   1:  PR[91,1] = PR[90,1] + -14.001;
   1:  PR[91,2] = PR[90,2] + -17.236;
   1:L PR[91] R[100]mm/sec CNT100;
   1:  PR[91,1] = PR[90,1] + -10.509;
   1:  PR[91,2] = PR[90,2] + -15.414;
   1:L PR[91] R[100]mm/sec CNT100;
   1:  PR[91,1] = PR[90,1] + -10.313;
   1:  PR[91,2] = PR[90,2] + -15.321;
   1:L PR[91] R[100]mm/sec CNT100;
   1:  PR[91,1] = PR[90,1] + -10.178;
   1:  PR[91,2] = PR[90,2] + -15.230;
   1:L PR[91] R[100]mm/sec CNT100;
   1:  PR[91,1] = PR[90,1] + -7.558;
   1:  PR[91,2] = PR[90,2] + -13.063;
   1:L PR[91] R[100]mm/sec CNT100;
   1:  PR[91,1] = PR[90,1] + -7.094;
   1:  PR[91,2] = PR[90,2] + -12.647;
   1:L PR[91] R[100]mm/sec CNT100;
   1:  PR[91,1] = PR[90,1] + -6.546;
   1:  PR[91,2] = PR[90,2] + -11.988;
   1:L PR[91] R[100]mm/sec CNT100;
   1:  PR[91,1] = PR[90,1] + -4.744;
   1:  PR[91,2] = PR[90,2] + -9.631;
   1:L PR[91] R[100]mm/sec CNT100;
   1:  PR[91,1] = PR[90,1] + -4.097;
   1:  PR[91,2] = PR[90,2] + -8.987;
   1:L PR[91] R[100]mm/sec CNT100;
   1:  PR[91,1] = PR[90,1] + -3.333;
   1:  PR[91,2] = PR[90,2] + -8.472;
   1:L PR[91] R[100]mm/sec CNT100;
   1:  PR[91,1] = PR[90,1] + -2.609;
   1:  PR[91,2] = PR[90,2] + -8.296;
   1:L PR[91] R[100]mm/sec CNT100;
   1:  PR[91,1] = PR[90,1] + -2.071;
   1:  PR[91,2] = PR[90,2] + -8.060;
   1:L PR[91] R[100]mm/sec CNT100;
   1:  PR[91,1] = PR[90,1] + 1.372;
   1:L PR[91] R[100]mm/sec CNT100;
   1:  PR[91,1] = PR[90,1] + 2.454;
   1:  PR[91,2] = PR[90,2] + -8.321;
   1:L PR[91] R[100]mm/sec CNT100;
   1:  PR[91,1] = PR[90,1] + 2.775;
   1:  PR[91,2] = PR[90,2] + -8.536;
   1:L PR[91] R[100]mm/sec CNT100;
   1:  PR[91,1] = PR[90,1] + 3.450;
   1:  PR[91,2] = PR[90,2] + -8.810;
   1:L PR[91] R[100]mm/sec CNT100;
   1:  PR[91,1] = PR[90,1] + 4.268;
   1:  PR[91,2] = PR[90,2] + -9.634;
   1:L PR[91] R[100]mm/sec CNT100;
   1:  PR[91,1] = PR[90,1] + 6.077;
   1:  PR[91,2] = PR[90,2] + -11.995;
   1:L PR[91] R[100]mm/sec CNT100;
   1:  PR[91,1] = PR[90,1] + 6.604;
   1:  PR[91,2] = PR[90,2] + -12.629;
   1:L PR[91] R[100]mm/sec CNT100;
   1:  PR[91,1] = PR[90,1] + 9.392;
   1:  PR[91,2] = PR[90,2] + -14.954;
   1:L PR[91] R[100]mm/sec CNT100;
   1:  PR[91,1] = PR[90,1] + 9.744;
   1:  PR[91,2] = PR[90,2] + -15.265;
   1:L PR[91] R[100]mm/sec CNT100;
   1:  PR[91,1] = PR[90,1] + 9.873;
   1:  PR[91,2] = PR[90,2] + -15.351;
   1:L PR[91] R[100]mm/sec CNT100;
   1:  PR[91,1] = PR[90,1] + 13.005;
   1:  PR[91,2] = PR[90,2] + -16.954;
   1:L PR[91] R[100]mm/sec CNT100;
   1:  PR[91,1] = PR[90,1] + 13.545;
   1:  PR[91,2] = PR[90,2] + -17.243;
   1:L PR[91] R[100]mm/sec CNT100;
   1:  PR[91,1] = PR[90,1] + 17.419;
   1:  PR[91,2] = PR[90,2] + -18.355;
   1:L PR[91] R[100]mm/sec CNT100;
   1:  PR[91,1] = PR[90,1] + 18.185;
   1:  PR[91,2] = PR[90,2] + -18.441;
   1:L PR[91] R[100]mm/sec CNT100;
   1:  PR[91,1] = PR[90,1] + 21.425;
   1:  PR[91,2] = PR[90,2] + -18.650;
   1:L PR[91] R[100]mm/sec CNT100;
   1:  PR[91,1] = PR[90,1] + 22.997;
   1:  PR[91,2] = PR[90,2] + -18.479;
   1:L PR[91] R[100]mm/sec CNT100;
   1:  PR[91,1] = PR[90,1] + 25.448;
   1:  PR[91,2] = PR[90,2] + -18.112;
   1:L PR[91] R[100]mm/sec CNT100;
   1:  PR[91,1] = PR[90,1] + 27.611;
   1:  PR[91,2] = PR[90,2] + -17.377;
   1:L PR[91] R[100]mm/sec CNT100;
   1:  PR[91,1] = PR[90,1] + 29.297;
   1:  PR[91,2] = PR[90,2] + -16.739;
   1:L PR[91] R[100]mm/sec CNT100;
   1:  PR[91,1] = PR[90,1] + 31.732;
   1:  PR[91,2] = PR[90,2] + -15.254;
   1:L PR[91] R[100]mm/sec CNT100;
   1:  PR[91,1] = PR[90,1] + 32.770;
   1:  PR[91,2] = PR[90,2] + -14.580;
   1:L PR[91] R[100]mm/sec CNT100;
   1:  PR[91,1] = PR[90,1] + 35.120;
   1:  PR[91,2] = PR[90,2] + -12.291;
   1:L PR[91] R[100]mm/sec CNT100;
   1:  PR[91,1] = PR[90,1] + 35.686;
   1:  PR[91,2] = PR[90,2] + -11.714;
   1:L PR[91] R[100]mm/sec CNT100;
   1:  PR[91,1] = PR[90,1] + 37.625;
   1:  PR[91,2] = PR[90,2] + -8.701;
   1:L PR[91] R[100]mm/sec CNT100;
   1:  PR[91,1] = PR[90,1] + 37.894;
   1:  PR[91,2] = PR[90,2] + -8.268;
   1:L PR[91] R[100]mm/sec CNT100;
   1:  PR[91,1] = PR[90,1] + 39.268;
   1:  PR[91,2] = PR[90,2] + -4.483;
   1:L PR[91] R[100]mm/sec CNT100;
   1:  PR[91,1] = PR[90,1] + 39.742;
   1:  PR[91,2] = PR[90,2] + -0.424;
   1:L PR[91] R[100]mm/sec CNT100;
   1:  PR[91,1] = PR[90,1] + 39.268;
   1:  PR[91,2] = PR[90,2] + 3.636;
   1:L PR[91] R[100]mm/sec CNT100;
   1:  PR[91,1] = PR[90,1] + 37.894;
   1:  PR[91,2] = PR[90,2] + 7.421;
   1:L PR[91] R[100]mm/sec CNT100;
   1:  PR[91,1] = PR[90,1] + 37.625;
   1:  PR[91,2] = PR[90,2] + 7.855;
   1:L PR[91] R[100]mm/sec CNT100;
   1:  PR[91,1] = PR[90,1] + 35.685;
   1:  PR[91,2] = PR[90,2] + 10.868;
   1:L PR[91] R[100]mm/sec CNT100;
   1:  PR[91,1] = PR[90,1] + 35.119;
   1:  PR[91,2] = PR[90,2] + 11.445;
   1:L PR[91] R[100]mm/sec CNT100;
   1:  PR[91,1] = PR[90,1] + 32.769;
   1:  PR[91,2] = PR[90,2] + 13.734;
   1:L PR[91] R[100]mm/sec CNT100;
   1:  PR[91,1] = PR[90,1] + 31.731;
   1:  PR[91,2] = PR[90,2] + 14.407;
   1:L PR[91] R[100]mm/sec CNT100;
   1:  PR[91,1] = PR[90,1] + 29.296;
   1:  PR[91,2] = PR[90,2] + 15.893;
   1:L PR[91] R[100]mm/sec CNT100;
   1:  PR[91,1] = PR[90,1] + 27.609;
   1:  PR[91,2] = PR[90,2] + 16.530;
   1:L PR[91] R[100]mm/sec CNT100;
   1:  PR[91,1] = PR[90,1] + 25.447;
   1:  PR[91,2] = PR[90,2] + 17.265;
   1:L PR[91] R[100]mm/sec CNT100;
   1:  PR[91,1] = PR[90,1] + 22.996;
   1:  PR[91,2] = PR[90,2] + 17.632;
   1:L PR[91] R[100]mm/sec CNT100;
   1:  PR[91,1] = PR[90,1] + 21.423;
   1:  PR[91,2] = PR[90,2] + 17.802;
   1:L PR[91] R[100]mm/sec CNT100;
   1:  PR[91,1] = PR[90,1] + 18.184;
   1:  PR[91,2] = PR[90,2] + 17.594;
   1:L PR[91] R[100]mm/sec CNT100;
   1:  PR[91,1] = PR[90,1] + 17.418;
   1:  PR[91,2] = PR[90,2] + 17.508;
   1:L PR[91] R[100]mm/sec CNT100;
   1:  PR[91,1] = PR[90,1] + 13.543;
   1:  PR[91,2] = PR[90,2] + 16.395;
   1:L PR[91] R[100]mm/sec CNT100;
   1:  PR[91,1] = PR[90,1] + 13.009;
   1:  PR[91,2] = PR[90,2] + 16.109;
   1:L PR[91] R[100]mm/sec CNT100;
   1:  PR[91,1] = PR[90,1] + 10.031;
   1:  PR[91,2] = PR[90,2] + 14.572;
   1:L PR[91] R[100]mm/sec CNT100;
   1:  PR[91,1] = PR[90,1] + 9.841;
   1:  PR[91,2] = PR[90,2] + 14.482;
   1:L PR[91] R[100]mm/sec CNT100;
   1:  PR[91,1] = PR[90,1] + 9.711;
   1:  PR[91,2] = PR[90,2] + 14.396;
   1:L PR[91] R[100]mm/sec CNT100;
   1:  PR[91,1] = PR[90,1] + 7.091;
   1:  PR[91,2] = PR[90,2] + 12.226;
   1:L PR[91] R[100]mm/sec CNT100;
   1:  PR[91,1] = PR[90,1] + 6.630;
   1:  PR[91,2] = PR[90,2] + 11.813;
   1:L PR[91] R[100]mm/sec CNT100;
   1:  PR[91,1] = PR[90,1] + 6.077;
   1:  PR[91,2] = PR[90,2] + 11.147;
   1:L PR[91] R[100]mm/sec CNT100;
   1:  PR[91,1] = PR[90,1] + 4.268;
   1:  PR[91,2] = PR[90,2] + 8.785;
   1:L PR[91] R[100]mm/sec CNT100;
   1:  PR[91,1] = PR[90,1] + 3.627;
   1:  PR[91,2] = PR[90,2] + 8.142;
   1:L PR[91] R[100]mm/sec CNT100;
   1:  PR[91,1] = PR[90,1] + 2.859;
   1:  PR[91,2] = PR[90,2] + 7.624;
   1:L PR[91] R[100]mm/sec CNT100;
   1:  PR[91,1] = PR[90,1] + 2.132;
   1:  PR[91,2] = PR[90,2] + 7.448;
   1:L PR[91] R[100]mm/sec CNT100;
   1:  PR[91,1] = PR[90,1] + 1.592;
   1:  PR[91,2] = PR[90,2] + 7.213;
   1:L PR[91] R[100]mm/sec CNT100;
   1:  PR[91] = PR[90];
   1:  PR[91,1] = PR[90,1] + -1.650;
   1:  PR[91,2] = PR[90,2] + 7.757;
   1:  PR[91,3] = PR[90,3] + 20.995;
   1:L PR[91] R[100]mm/sec CNT100;
   1:  PR[91,1] = PR[90,1] + -2.898;
   1:  PR[91,2] = PR[90,2] + 8.058;
   1:L PR[91] R[100]mm/sec CNT100;
   1:  PR[91,1] = PR[90,1] + -3.294;
   1:  PR[91,2] = PR[90,2] + 8.324;
   1:L PR[91] R[100]mm/sec CNT100;
   1:  PR[91,1] = PR[90,1] + -3.766;
   1:  PR[91,2] = PR[90,2] + 8.516;
   1:L PR[91] R[100]mm/sec CNT100;
   1:  PR[91,1] = PR[90,1] + -4.523;
   1:  PR[91,2] = PR[90,2] + 9.302;
   1:L PR[91] R[100]mm/sec CNT100;
   1:  PR[91,1] = PR[90,1] + -5.363;
   1:  PR[91,2] = PR[90,2] + 10.400;
   1:L PR[91] R[100]mm/sec CNT100;
   1:  PR[91,1] = PR[90,1] + -6.566;
   1:  PR[91,2] = PR[90,2] + 11.846;
   1:L PR[91] R[100]mm/sec CNT100;
   1:  PR[91,1] = PR[90,1] + -8.018;
   1:  PR[91,2] = PR[90,2] + 13.056;
   1:L PR[91] R[100]mm/sec CNT100;
   1:  PR[91,1] = PR[90,1] + -9.282;
   1:  PR[91,2] = PR[90,2] + 14.171;
   1:L PR[91] R[100]mm/sec CNT100;
   1:  PR[91,1] = PR[90,1] + -10.188;
   1:  PR[91,2] = PR[90,2] + 14.780;
   1:L PR[91] R[100]mm/sec CNT100;
   1:  PR[91,1] = PR[90,1] + -12.854;
   1:  PR[91,2] = PR[90,2] + 16.148;
   1:L PR[91] R[100]mm/sec CNT100;
   1:  PR[91,1] = PR[90,1] + -13.521;
   1:  PR[91,2] = PR[90,2] + 16.470;
   1:L PR[91] R[100]mm/sec CNT100;
   1:  PR[91,1] = PR[90,1] + -13.956;
   1:  PR[91,2] = PR[90,2] + 16.611;
   1:L PR[91] R[100]mm/sec CNT100;
   1:  PR[91,1] = PR[90,1] + -17.655;
   1:  PR[91,2] = PR[90,2] + 17.601;
   1:L PR[91] R[100]mm/sec CNT100;
   1:  PR[91,1] = PR[90,1] + -18.894;
   1:  PR[91,2] = PR[90,2] + 17.666;
   1:L PR[91] R[100]mm/sec CNT100;
   1:  PR[91,1] = PR[90,1] + -21.828;
   1:  PR[91,2] = PR[90,2] + 17.855;
   1:L PR[91] R[100]mm/sec CNT100;
   1:  PR[91,1] = PR[90,1] + -22.170;
   1:  PR[91,2] = PR[90,2] + 17.818;
   1:L PR[91] R[100]mm/sec CNT100;
   1:  PR[91,1] = PR[90,1] + -25.820;
   1:  PR[91,2] = PR[90,2] + 17.274;
   1:L PR[91] R[100]mm/sec CNT100;
   1:  PR[91,1] = PR[90,1] + -26.878;
   1:  PR[91,2] = PR[90,2] + 16.914;
   1:L PR[91] R[100]mm/sec CNT100;
   1:  PR[91,1] = PR[90,1] + -29.633;
   1:  PR[91,2] = PR[90,2] + 15.872;
   1:L PR[91] R[100]mm/sec CNT100;
   1:  PR[91,1] = PR[90,1] + -31.131;
   1:  PR[91,2] = PR[90,2] + 14.957;
   1:L PR[91] R[100]mm/sec CNT100;
   1:  PR[91,1] = PR[90,1] + -33.074;
   1:  PR[91,2] = PR[90,2] + 13.696;
   1:L PR[91] R[100]mm/sec CNT100;
   1:  PR[91,1] = PR[90,1] + -34.682;
   1:  PR[91,2] = PR[90,2] + 12.133;
   1:L PR[91] R[100]mm/sec CNT100;
   1:  PR[91,1] = PR[90,1] + -35.960;
   1:  PR[91,2] = PR[90,2] + 10.834;
   1:L PR[91] R[100]mm/sec CNT100;
   1:  PR[91,1] = PR[90,1] + -37.364;
   1:  PR[91,2] = PR[90,2] + 8.651;
   1:L PR[91] R[100]mm/sec CNT100;
   1:  PR[91,1] = PR[90,1] + -38.143;
   1:  PR[91,2] = PR[90,2] + 7.394;
   1:L PR[91] R[100]mm/sec CNT100;
   1:  PR[91,1] = PR[90,1] + -39.504;
   1:  PR[91,2] = PR[90,2] + 3.616;
   1:L PR[91] R[100]mm/sec CNT100;
   1:  PR[91,1] = PR[90,1] + -39.844;
   1:  PR[91,2] = PR[90,2] + 0.678;
   1:L PR[91] R[100]mm/sec CNT100;
   1:  PR[91,1] = PR[90,1] + -39.986;
   1:  PR[91,2] = PR[90,2] + -0.438;
   1:L PR[91] R[100]mm/sec CNT100;
   1:  PR[91,1] = PR[90,1] + -39.718;
   1:  PR[91,2] = PR[90,2] + -2.762;
   1:L PR[91] R[100]mm/sec CNT100;
   1:  PR[91,1] = PR[90,1] + -39.636;
   1:  PR[91,2] = PR[90,2] + -3.261;
   1:L PR[91] R[100]mm/sec CNT100;
   1:  PR[91,1] = PR[90,1] + -39.501;
   1:  PR[91,2] = PR[90,2] + -4.475;
   1:L PR[91] R[100]mm/sec CNT100;
   1:  PR[91,1] = PR[90,1] + -39.096;
   1:  PR[91,2] = PR[90,2] + -5.618;
   1:L PR[91] R[100]mm/sec CNT100;
   1:  PR[91,1] = PR[90,1] + -38.145;
   1:  PR[91,2] = PR[90,2] + -8.239;
   1:L PR[91] R[100]mm/sec CNT100;
   1:  PR[91,1] = PR[90,1] + -37.364;
   1:  PR[91,2] = PR[90,2] + -9.499;
   1:L PR[91] R[100]mm/sec CNT100;
   1:  PR[91,1] = PR[90,1] + -35.960;
   1:  PR[91,2] = PR[90,2] + -11.682;
   1:L PR[91] R[100]mm/sec CNT100;
   1:  PR[91,1] = PR[90,1] + -34.681;
   1:  PR[91,2] = PR[90,2] + -12.981;
   1:L PR[91] R[100]mm/sec CNT100;
   1:  PR[91,1] = PR[90,1] + -33.073;
   1:  PR[91,2] = PR[90,2] + -14.545;
   1:L PR[91] R[100]mm/sec CNT100;
   1:  PR[91,1] = PR[90,1] + -31.128;
   1:  PR[91,2] = PR[90,2] + -15.806;
   1:L PR[91] R[100]mm/sec CNT100;
   1:  PR[91,1] = PR[90,1] + -29.631;
   1:  PR[91,2] = PR[90,2] + -16.720;
   1:L PR[91] R[100]mm/sec CNT100;
   1:  PR[91,1] = PR[90,1] + -26.874;
   1:  PR[91,2] = PR[90,2] + -17.763;
   1:L PR[91] R[100]mm/sec CNT100;
   1:  PR[91,1] = PR[90,1] + -25.817;
   1:  PR[91,2] = PR[90,2] + -18.122;
   1:L PR[91] R[100]mm/sec CNT100;
   1:  PR[91,1] = PR[90,1] + -22.165;
   1:  PR[91,2] = PR[90,2] + -18.666;
   1:L PR[91] R[100]mm/sec CNT100;
   1:  PR[91,1] = PR[90,1] + -21.823;
   1:  PR[91,2] = PR[90,2] + -18.703;
   1:L PR[91] R[100]mm/sec CNT100;
   1:  PR[91,1] = PR[90,1] + -18.895;
   1:  PR[91,2] = PR[90,2] + -18.513;
   1:L PR[91] R[100]mm/sec CNT100;
   1:  PR[91,1] = PR[90,1] + -17.649;
   1:  PR[91,2] = PR[90,2] + -18.447;
   1:L PR[91] R[100]mm/sec CNT100;
   1:  PR[91,1] = PR[90,1] + -13.952;
   1:  PR[91,2] = PR[90,2] + -17.457;
   1:L PR[91] R[100]mm/sec CNT100;
   1:  PR[91,1] = PR[90,1] + -13.548;
   1:  PR[91,2] = PR[90,2] + -17.326;
   1:L PR[91] R[100]mm/sec CNT100;
   1:  PR[91,1] = PR[90,1] + -10.983;
   1:  PR[91,2] = PR[90,2] + -15.997;
   1:L PR[91] R[100]mm/sec CNT100;
   1:  PR[91,1] = PR[90,1] + -10.153;
   1:  PR[91,2] = PR[90,2] + -15.604;
   1:L PR[91] R[100]mm/sec CNT100;
   1:  PR[91,1] = PR[90,1] + -9.246;
   1:  PR[91,2] = PR[90,2] + -14.994;
   1:L PR[91] R[100]mm/sec CNT100;
   1:  PR[91,1] = PR[90,1] + -7.675;
   1:  PR[91,2] = PR[90,2] + -13.694;
   1:L PR[91] R[100]mm/sec CNT100;
   1:  PR[91,1] = PR[90,1] + -6.591;
   1:  PR[91,2] = PR[90,2] + -12.724;
   1:L PR[91] R[100]mm/sec CNT100;
   1:  PR[91,1] = PR[90,1] + -5.362;
   1:  PR[91,2] = PR[90,2] + -11.246;
   1:L PR[91] R[100]mm/sec CNT100;
   1:  PR[91,1] = PR[90,1] + -4.523;
   1:  PR[91,2] = PR[90,2] + -10.149;
   1:L PR[91] R[100]mm/sec CNT100;
   1:  PR[91,1] = PR[90,1] + -3.941;
   1:  PR[91,2] = PR[90,2] + -9.546;
   1:L PR[91] R[100]mm/sec CNT100;
   1:  PR[91,1] = PR[90,1] + -3.105;
   1:  PR[91,2] = PR[90,2] + -8.982;
   1:L PR[91] R[100]mm/sec CNT100;
   1:  PR[91,1] = PR[90,1] + -2.261;
   1:  PR[91,2] = PR[90,2] + -8.777;
   1:L PR[91] R[100]mm/sec CNT100;
   1:  PR[91,1] = PR[90,1] + -1.869;
   1:  PR[91,2] = PR[90,2] + -8.605;
   1:L PR[91] R[100]mm/sec CNT100;
   1:  PR[91,1] = PR[90,1] + 1.175;
   1:L PR[91] R[100]mm/sec CNT100;
   1:  PR[91,1] = PR[90,1] + 2.438;
   1:  PR[91,2] = PR[90,2] + -8.909;
   1:L PR[91] R[100]mm/sec CNT100;
   1:  PR[91,1] = PR[90,1] + 2.840;
   1:  PR[91,2] = PR[90,2] + -9.178;
   1:L PR[91] R[100]mm/sec CNT100;
   1:  PR[91,1] = PR[90,1] + 3.295;
   1:  PR[91,2] = PR[90,2] + -9.363;
   1:L PR[91] R[100]mm/sec CNT100;
   1:  PR[91,1] = PR[90,1] + 4.050;
   1:  PR[91,2] = PR[90,2] + -10.150;
   1:L PR[91] R[100]mm/sec CNT100;
   1:  PR[91,1] = PR[90,1] + 4.893;
   1:  PR[91,2] = PR[90,2] + -11.249;
   1:L PR[91] R[100]mm/sec CNT100;
   1:  PR[91,1] = PR[90,1] + 6.106;
   1:  PR[91,2] = PR[90,2] + -12.710;
   1:L PR[91] R[100]mm/sec CNT100;
   1:  PR[91,1] = PR[90,1] + 7.561;
   1:  PR[91,2] = PR[90,2] + -13.924;
   1:L PR[91] R[100]mm/sec CNT100;
   1:  PR[91,1] = PR[90,1] + 8.816;
   1:  PR[91,2] = PR[90,2] + -15.032;
   1:L PR[91] R[100]mm/sec CNT100;
   1:  PR[91,1] = PR[90,1] + 9.709;
   1:  PR[91,2] = PR[90,2] + -15.631;
   1:L PR[91] R[100]mm/sec CNT100;
   1:  PR[91,1] = PR[90,1] + 12.375;
   1:  PR[91,2] = PR[90,2] + -16.995;
   1:L PR[91] R[100]mm/sec CNT100;
   1:  PR[91,1] = PR[90,1] + 13.041;
   1:  PR[91,2] = PR[90,2] + -17.316;
   1:L PR[91] R[100]mm/sec CNT100;
   1:  PR[91,1] = PR[90,1] + 13.479;
   1:  PR[91,2] = PR[90,2] + -17.458;
   1:L PR[91] R[100]mm/sec CNT100;
   1:  PR[91,1] = PR[90,1] + 17.181;
   1:  PR[91,2] = PR[90,2] + -18.448;
   1:L PR[91] R[100]mm/sec CNT100;
   1:  PR[91,1] = PR[90,1] + 18.414;
   1:  PR[91,2] = PR[90,2] + -18.514;
   1:L PR[91] R[100]mm/sec CNT100;
   1:  PR[91,1] = PR[90,1] + 21.352;
   1:  PR[91,2] = PR[90,2] + -18.703;
   1:L PR[91] R[100]mm/sec CNT100;
   1:  PR[91,1] = PR[90,1] + 21.695;
   1:  PR[91,2] = PR[90,2] + -18.666;
   1:L PR[91] R[100]mm/sec CNT100;
   1:  PR[91,1] = PR[90,1] + 25.343;
   1:  PR[91,2] = PR[90,2] + -18.119;
   1:L PR[91] R[100]mm/sec CNT100;
   1:  PR[91,1] = PR[90,1] + 26.401;
   1:  PR[91,2] = PR[90,2] + -17.760;
   1:L PR[91] R[100]mm/sec CNT100;
   1:  PR[91,1] = PR[90,1] + 29.155;
   1:  PR[91,2] = PR[90,2] + -16.718;
   1:L PR[91] R[100]mm/sec CNT100;
   1:  PR[91,1] = PR[90,1] + 30.653;
   1:  PR[91,2] = PR[90,2] + -15.804;
   1:L PR[91] R[100]mm/sec CNT100;
   1:  PR[91,1] = PR[90,1] + 32.594;
   1:  PR[91,2] = PR[90,2] + -14.546;
   1:L PR[91] R[100]mm/sec CNT100;
   1:  PR[91,1] = PR[90,1] + 34.201;
   1:  PR[91,2] = PR[90,2] + -12.981;
   1:L PR[91] R[100]mm/sec CNT100;
   1:  PR[91,1] = PR[90,1] + 35.480;
   1:  PR[91,2] = PR[90,2] + -11.676;
   1:L PR[91] R[100]mm/sec CNT100;
   1:  PR[91,1] = PR[90,1] + 36.886;
   1:  PR[91,2] = PR[90,2] + -9.492;
   1:L PR[91] R[100]mm/sec CNT100;
   1:  PR[91,1] = PR[90,1] + 37.665;
   1:  PR[91,2] = PR[90,2] + -8.238;
   1:L PR[91] R[100]mm/sec CNT100;
   1:  PR[91,1] = PR[90,1] + 39.024;
   1:  PR[91,2] = PR[90,2] + -4.475;
   1:L PR[91] R[100]mm/sec CNT100;
   1:  PR[91,1] = PR[90,1] + 39.364;
   1:  PR[91,2] = PR[90,2] + -1.532;
   1:L PR[91] R[100]mm/sec CNT100;
   1:  PR[91,1] = PR[90,1] + 39.507;
   1:  PR[91,2] = PR[90,2] + -0.410;
   1:L PR[91] R[100]mm/sec CNT100;
   1:  PR[91,1] = PR[90,1] + 39.238;
   1:  PR[91,2] = PR[90,2] + 1.922;
   1:L PR[91] R[100]mm/sec CNT100;
   1:  PR[91,1] = PR[90,1] + 39.156;
   1:  PR[91,2] = PR[90,2] + 2.422;
   1:L PR[91] R[100]mm/sec CNT100;
   1:  PR[91,1] = PR[90,1] + 39.022;
   1:  PR[91,2] = PR[90,2] + 3.634;
   1:L PR[91] R[100]mm/sec CNT100;
   1:  PR[91,1] = PR[90,1] + 37.665;
   1:  PR[91,2] = PR[90,2] + 7.391;
   1:L PR[91] R[100]mm/sec CNT100;
   1:  PR[91,1] = PR[90,1] + 36.885;
   1:  PR[91,2] = PR[90,2] + 8.646;
   1:L PR[91] R[100]mm/sec CNT100;
   1:  PR[91,1] = PR[90,1] + 35.480;
   1:  PR[91,2] = PR[90,2] + 10.830;
   1:L PR[91] R[100]mm/sec CNT100;
   1:  PR[91,1] = PR[90,1] + 34.200;
   1:  PR[91,2] = PR[90,2] + 12.134;
